Yaskawa INFORM job: A_ROOF_UPPER_0614_2_PAINT_35.JBI

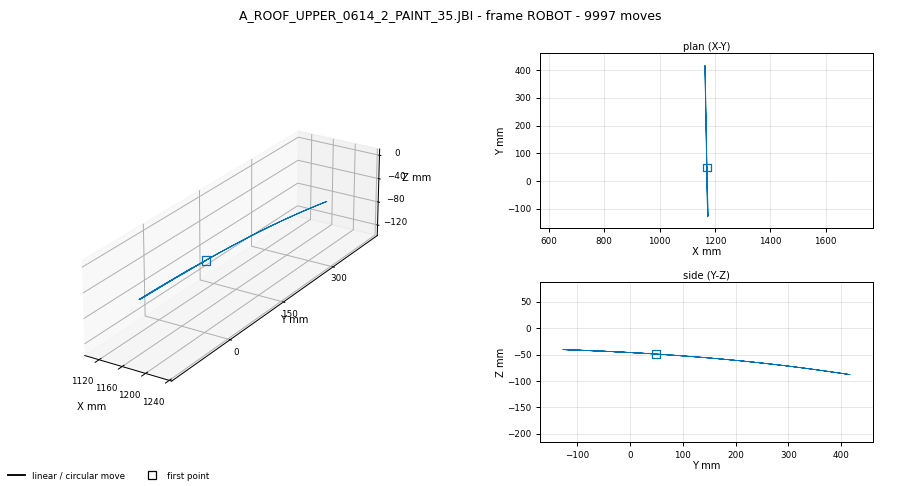
[picture p0: tool path of A_ROOF_UPPER_0614_2_PAINT_35.JBI in frame ROBOT, 9997 of 9997 moves have a stored position in this frame; points joined in program order, loops and branches not executed]
/JOB
//NAME A_ROOF_UPPER_0614_2_PAINT35
//POS
///NPOS 9997,0,0,0,0,0
///TOOL 1
///USER 0
///POSTYPE ROBOT
///RECTAN
///RCONF 1,0,0,0,0,0,0,0,0,0,0,0,0,0,0,0,0,0,0,0,0,0,0,0
C00000=1171.843,48.979,-48.682,-179.550,6.056,148.954
C00001=1171.848,48.730,-48.666,-179.552,6.054,148.954
C00002=1171.853,48.480,-48.650,-179.555,6.054,148.955
C00003=1171.858,48.231,-48.635,-179.557,6.053,148.955
C00004=1171.863,47.981,-48.619,-179.560,6.052,148.956
C00005=1171.868,47.732,-48.604,-179.562,6.051,148.956
C00006=1171.873,47.482,-48.588,-179.565,6.050,148.957
C00007=1171.878,47.233,-48.571,-179.568,6.049,148.958
C00008=1171.882,46.984,-48.556,-179.570,6.048,148.958
C00009=1171.888,46.734,-48.541,-179.573,6.048,148.959
C00010=1171.893,46.484,-48.525,-179.575,6.047,148.959
C00011=1171.898,46.235,-48.509,-179.578,6.046,148.960
C00012=1171.903,45.986,-48.494,-179.581,6.045,148.960
C00013=1171.908,45.736,-48.479,-179.583,6.044,148.961
C00014=1171.913,45.487,-48.462,-179.586,6.043,148.962
C00015=1171.918,45.237,-48.446,-179.589,6.042,148.962
C00016=1171.923,44.988,-48.431,-179.591,6.041,148.963
C00017=1171.927,44.738,-48.415,-179.593,6.041,148.963
C00018=1171.933,44.489,-48.400,-179.597,6.039,148.964
C00019=1171.938,44.239,-48.384,-179.599,6.038,148.964
C00020=1171.943,43.990,-48.369,-179.601,6.038,148.965
C00021=1171.948,43.740,-48.353,-179.604,6.036,148.966
C00022=1171.953,43.491,-48.338,-179.607,6.036,148.966
C00023=1171.958,43.242,-48.323,-179.609,6.035,148.967
C00024=1171.963,42.992,-48.307,-179.612,6.034,148.967
C00025=1171.968,42.742,-48.291,-179.614,6.033,148.968
C00026=1171.972,42.493,-48.276,-179.617,6.032,148.968
C00027=1171.978,42.244,-48.261,-179.620,6.032,148.969
C00028=1171.983,41.994,-48.245,-179.622,6.031,148.970
C00029=1171.988,41.745,-48.230,-179.625,6.030,148.970
C00030=1171.993,41.495,-48.214,-179.627,6.029,148.971
C00031=1171.998,41.246,-48.199,-179.630,6.028,148.971
C00032=1172.003,40.997,-48.184,-179.633,6.027,148.972
C00033=1172.008,40.747,-48.168,-179.635,6.026,148.972
C00034=1172.012,40.497,-48.153,-179.637,6.025,148.973
C00035=1172.018,40.247,-48.138,-179.640,6.025,148.974
C00036=1172.023,39.998,-48.122,-179.643,6.023,148.974
C00037=1172.028,39.749,-48.107,-179.645,6.023,148.975
C00038=1172.033,39.499,-48.092,-179.648,6.022,148.975
C00039=1172.039,39.250,-48.076,-179.650,6.021,148.976
C00040=1172.043,39.000,-48.061,-179.653,6.020,148.977
C00041=1172.048,38.751,-48.045,-179.656,6.019,148.977
C00042=1172.053,38.502,-48.030,-179.658,6.019,148.978
C00043=1172.058,38.252,-48.015,-179.661,6.018,148.978
C00044=1172.063,38.003,-48.000,-179.664,6.016,148.979
C00045=1172.068,37.753,-47.985,-179.666,6.016,148.979
C00046=1172.072,37.503,-47.969,-179.668,6.015,148.980
C00047=1172.078,37.254,-47.954,-179.671,6.015,148.981
C00048=1172.084,37.004,-47.939,-179.674,6.013,148.981
C00049=1172.088,36.755,-47.924,-179.677,6.012,148.982
C00050=1172.094,36.505,-47.908,-179.679,6.012,148.982
C00051=1172.098,36.256,-47.893,-179.681,6.011,148.983
C00052=1172.104,36.007,-47.878,-179.684,6.011,148.983
C00053=1172.109,35.757,-47.863,-179.687,6.009,148.984
C00054=1172.113,35.507,-47.847,-179.689,6.008,148.985
C00055=1172.118,35.258,-47.832,-179.691,6.008,148.985
C00056=1172.124,35.008,-47.817,-179.694,6.007,148.986
C00057=1172.128,34.759,-47.802,-179.697,6.006,148.986
C00058=1172.134,34.510,-47.787,-179.700,6.005,148.987
C00059=1172.138,34.260,-47.772,-179.702,6.004,148.988
C00060=1172.144,34.010,-47.757,-179.704,6.004,148.988
C00061=1172.149,33.761,-47.742,-179.707,6.003,148.989
C00062=1172.153,33.512,-47.727,-179.710,6.002,148.989
C00063=1172.159,33.262,-47.712,-179.712,6.001,148.990
C00064=1172.163,33.012,-47.697,-179.715,6.000,148.990
C00065=1172.169,32.763,-47.681,-179.717,6.000,148.991
C00066=1172.173,32.513,-47.667,-179.720,5.998,148.992
C00067=1172.179,32.264,-47.651,-179.723,5.997,148.992
C00068=1172.184,32.014,-47.637,-179.725,5.997,148.993
C00069=1172.188,31.765,-47.622,-179.728,5.996,148.993
C00070=1172.194,31.516,-47.607,-179.730,5.996,148.994
C00071=1172.199,31.266,-47.592,-179.733,5.994,148.994
C00072=1172.203,31.017,-47.577,-179.735,5.993,148.995
C00073=1172.209,30.767,-47.562,-179.738,5.993,148.996
C00074=1172.214,30.518,-47.547,-179.741,5.992,148.996
C00075=1172.219,30.268,-47.533,-179.743,5.992,148.997
C00076=1172.224,30.019,-47.518,-179.746,5.990,148.997
C00077=1172.229,29.769,-47.503,-179.748,5.989,148.998
C00078=1172.234,29.520,-47.488,-179.751,5.989,148.999
C00079=1172.239,29.271,-47.473,-179.754,5.988,148.999
C00080=1172.244,29.021,-47.458,-179.756,5.988,149.000
C00081=1172.249,28.771,-47.443,-179.759,5.986,149.000
C00082=1172.255,28.503,-47.427,-179.762,5.986,149.001
C00083=1172.260,28.234,-47.411,-179.764,5.985,149.001
C00084=1172.266,27.965,-47.395,-179.767,5.984,149.002
C00085=1172.271,27.696,-47.379,-179.770,5.983,149.003
C00086=1172.276,27.446,-47.365,-179.772,5.983,149.004
C00087=1172.281,27.197,-47.350,-179.774,5.982,149.004
C00088=1172.286,26.947,-47.335,-179.777,5.981,149.005
C00089=1172.291,26.697,-47.321,-179.780,5.980,149.005
C00090=1172.296,26.448,-47.305,-179.782,5.979,149.006
C00091=1172.301,26.198,-47.291,-179.785,5.979,149.006
C00092=1172.306,25.949,-47.276,-179.787,5.978,149.007
C00093=1172.311,25.699,-47.262,-179.790,5.977,149.008
C00094=1172.317,25.449,-47.247,-179.792,5.977,149.008
C00095=1172.321,25.200,-47.232,-179.795,5.975,149.009
C00096=1172.326,24.951,-47.218,-179.798,5.975,149.009
C00097=1172.331,24.702,-47.203,-179.800,5.974,149.010
C00098=1172.337,24.452,-47.188,-179.803,5.974,149.011
C00099=1172.342,24.203,-47.174,-179.805,5.973,149.011
C00100=1172.347,23.953,-47.159,-179.808,5.972,149.012
C00101=1172.352,23.704,-47.145,-179.811,5.971,149.012
C00102=1172.357,23.454,-47.130,-179.813,5.970,149.013
C00103=1172.362,23.204,-47.115,-179.816,5.970,149.013
C00104=1172.367,22.955,-47.100,-179.818,5.969,149.014
C00105=1172.372,22.705,-47.086,-179.820,5.968,149.015
C00106=1172.377,22.455,-47.072,-179.823,5.968,149.015
C00107=1172.382,22.206,-47.057,-179.826,5.966,149.016
C00108=1172.386,21.957,-47.043,-179.829,5.966,149.016
C00109=1172.392,21.707,-47.028,-179.831,5.965,149.017
C00110=1172.398,21.458,-47.014,-179.833,5.964,149.018
C00111=1172.402,21.209,-46.999,-179.836,5.964,149.018
C00112=1172.407,20.959,-46.985,-179.838,5.963,149.019
C00113=1172.412,20.709,-46.970,-179.841,5.962,149.019
C00114=1172.417,20.459,-46.956,-179.844,5.961,149.020
C00115=1172.422,20.210,-46.942,-179.846,5.960,149.021
C00116=1172.427,19.961,-46.927,-179.849,5.960,149.021
C00117=1172.433,19.711,-46.912,-179.851,5.959,149.022
C00118=1172.438,19.462,-46.898,-179.854,5.959,149.022
C00119=1172.443,19.212,-46.884,-179.856,5.958,149.023
C00120=1172.448,18.962,-46.869,-179.858,5.957,149.023
C00121=1172.453,18.712,-46.855,-179.862,5.956,149.024
C00122=1172.458,18.463,-46.840,-179.864,5.955,149.025
C00123=1172.463,18.214,-46.826,-179.867,5.955,149.025
C00124=1172.468,17.965,-46.812,-179.869,5.954,149.026
C00125=1172.473,17.715,-46.798,-179.871,5.953,149.026
C00126=1172.478,17.465,-46.783,-179.874,5.953,149.027
C00127=1172.483,17.216,-46.769,-179.876,5.952,149.028
C00128=1172.488,16.966,-46.755,-179.879,5.951,149.028
C00129=1172.493,16.716,-46.741,-179.881,5.951,149.029
C00130=1172.498,16.467,-46.727,-179.884,5.949,149.029
C00131=1172.503,16.217,-46.712,-179.887,5.949,149.030
C00132=1172.508,15.968,-46.698,-179.889,5.948,149.031
C00133=1172.513,15.719,-46.683,-179.892,5.948,149.031
C00134=1172.518,15.469,-46.669,-179.894,5.947,149.032
C00135=1172.524,15.220,-46.655,-179.896,5.946,149.032
C00136=1172.528,14.970,-46.641,-179.899,5.946,149.033
C00137=1172.533,14.720,-46.626,-179.902,5.945,149.034
C00138=1172.538,14.471,-46.612,-179.904,5.944,149.034
C00139=1172.544,14.222,-46.598,-179.907,5.943,149.035
C00140=1172.549,13.972,-46.584,-179.909,5.942,149.035
C00141=1172.554,13.722,-46.570,-179.912,5.942,149.036
C00142=1172.559,13.473,-46.555,-179.915,5.941,149.037
C00143=1172.565,13.223,-46.542,-179.917,5.941,149.037
C00144=1172.570,12.973,-46.528,-179.919,5.940,149.038
C00145=1172.575,12.724,-46.514,-179.922,5.940,149.038
C00146=1172.580,12.474,-46.499,-179.924,5.939,149.039
C00147=1172.585,12.225,-46.485,-179.927,5.938,149.040
C00148=1172.590,11.975,-46.471,-179.929,5.937,149.040
C00149=1172.595,11.725,-46.457,-179.932,5.936,149.041
C00150=1172.600,11.476,-46.443,-179.935,5.936,149.041
C00151=1172.606,11.227,-46.429,-179.937,5.935,149.042
C00152=1172.610,10.977,-46.415,-179.940,5.934,149.043
C00153=1172.615,10.728,-46.401,-179.942,5.934,149.043
C00154=1172.620,10.477,-46.387,-179.945,5.933,149.044
C00155=1172.626,10.228,-46.373,-179.947,5.933,149.044
C00156=1172.630,9.979,-46.359,-179.949,5.932,149.045
C00157=1172.635,9.729,-46.345,-179.952,5.931,149.046
C00158=1172.641,9.480,-46.331,-179.955,5.931,149.046
C00159=1172.646,9.230,-46.317,-179.957,5.930,149.047
C00160=1172.650,8.980,-46.304,-179.960,5.929,149.047
C00161=1172.656,8.731,-46.290,-179.963,5.928,149.048
C00162=1172.661,8.481,-46.275,-179.965,5.927,149.049
C00163=1172.666,8.232,-46.261,-179.968,5.927,149.049
C00164=1172.671,7.983,-46.247,-179.970,5.926,149.050
C00165=1172.676,7.733,-46.234,-179.972,5.926,149.050
C00166=1172.681,7.483,-46.220,-179.975,5.925,149.051
C00167=1172.687,7.234,-46.206,-179.977,5.924,149.052
C00168=1172.691,6.984,-46.192,-179.980,5.924,149.052
C00169=1172.697,6.734,-46.178,-179.983,5.923,149.053
C00170=1172.702,6.485,-46.165,-179.985,5.923,149.053
C00171=1172.706,6.235,-46.151,-179.987,5.922,149.054
C00172=1172.711,5.986,-46.136,-179.990,5.921,149.054
C00173=1172.717,5.736,-46.123,-179.992,5.921,149.055
C00174=1172.722,5.486,-46.109,-179.995,5.920,149.056
C00175=1172.726,5.237,-46.095,-179.997,5.919,149.056
C00176=1172.732,4.987,-46.082,-180.000,5.919,149.057
C00177=1172.737,4.738,-46.068,179.997,5.918,149.058
C00178=1172.743,4.489,-46.054,179.995,5.917,149.058
C00179=1172.747,4.239,-46.041,179.992,5.916,149.059
C00180=1172.752,3.989,-46.027,179.990,5.916,149.059
C00181=1172.758,3.740,-46.013,179.987,5.915,149.060
C00182=1172.762,3.490,-46.000,179.985,5.915,149.061
C00183=1172.768,3.241,-45.986,179.983,5.914,149.061
C00184=1172.773,2.991,-45.972,179.980,5.913,149.062
C00185=1172.778,2.741,-45.958,179.977,5.913,149.063
C00186=1172.783,2.472,-45.944,179.975,5.912,149.063
C00187=1172.789,2.203,-45.929,179.972,5.912,149.064
C00188=1172.794,1.934,-45.914,179.970,5.911,149.064
C00189=1172.800,1.664,-45.899,179.967,5.910,149.065
C00190=1172.806,1.415,-45.886,179.964,5.909,149.066
C00191=1172.810,1.165,-45.872,179.962,5.909,149.066
C00192=1172.816,0.916,-45.859,179.959,5.908,149.067
C00193=1172.821,0.666,-45.845,179.956,5.908,149.068
C00194=1172.826,0.417,-45.832,179.954,5.907,149.068
C00195=1172.831,0.167,-45.818,179.952,5.906,149.069
C00196=1172.835,-0.083,-45.805,179.949,5.905,149.069
C00197=1172.841,-0.332,-45.791,179.947,5.905,149.070
C00198=1172.846,-0.583,-45.777,179.944,5.905,149.071
C00199=1172.851,-0.831,-45.764,179.942,5.904,149.071
C00200=1172.856,-1.082,-45.750,179.939,5.903,149.072
C00201=1172.862,-1.331,-45.736,179.937,5.903,149.072
C00202=1172.866,-1.581,-45.723,179.934,5.902,149.073
C00203=1172.872,-1.830,-45.710,179.932,5.902,149.074
C00204=1172.876,-2.080,-45.697,179.929,5.901,149.074
C00205=1172.882,-2.329,-45.683,179.927,5.900,149.075
C00206=1172.886,-2.579,-45.670,179.924,5.900,149.075
C00207=1172.892,-2.828,-45.657,179.922,5.899,149.076
C00208=1172.897,-3.078,-45.642,179.920,5.898,149.077
C00209=1172.902,-3.327,-45.630,179.917,5.898,149.077
C00210=1172.907,-3.577,-45.615,179.915,5.897,149.078
C00211=1172.912,-3.826,-45.603,179.912,5.897,149.078
C00212=1172.918,-4.077,-45.589,179.909,5.896,149.079
C00213=1172.923,-4.325,-45.576,179.907,5.895,149.080
C00214=1172.928,-4.576,-45.562,179.905,5.895,149.080
C00215=1172.933,-4.825,-45.550,179.902,5.895,149.081
C00216=1172.938,-5.075,-45.535,179.900,5.894,149.081
C00217=1172.943,-5.324,-45.523,179.897,5.893,149.082
C00218=1172.948,-5.574,-45.509,179.895,5.892,149.083
C00219=1172.953,-5.823,-45.496,179.892,5.892,149.083
C00220=1172.959,-6.073,-45.483,179.890,5.891,149.084
C00221=1172.963,-6.323,-45.470,179.887,5.891,149.084
C00222=1172.969,-6.572,-45.456,179.885,5.890,149.085
C00223=1172.974,-6.822,-45.443,179.882,5.890,149.086
C00224=1172.979,-7.071,-45.430,179.880,5.889,149.086
C00225=1172.984,-7.321,-45.417,179.877,5.888,149.087
C00226=1172.989,-7.570,-45.403,179.875,5.888,149.088
C00227=1172.994,-7.820,-45.390,179.872,5.887,149.088
C00228=1173.000,-8.070,-45.377,179.870,5.887,149.089
C00229=1173.005,-8.319,-45.364,179.867,5.886,149.089
C00230=1173.009,-8.569,-45.350,179.865,5.885,149.090
C00231=1173.015,-8.818,-45.337,179.862,5.885,149.091
C00232=1173.020,-9.068,-45.324,179.860,5.884,149.091
C00233=1173.025,-9.318,-45.311,179.857,5.884,149.092
C00234=1173.030,-9.567,-45.298,179.855,5.883,149.092
C00235=1173.035,-9.817,-45.285,179.853,5.882,149.093
C00236=1173.041,-10.066,-45.272,179.850,5.882,149.094
C00237=1173.045,-10.316,-45.259,179.847,5.881,149.094
C00238=1173.051,-10.566,-45.245,179.845,5.881,149.095
C00239=1173.056,-10.815,-45.233,179.842,5.880,149.095
C00240=1173.060,-11.065,-45.219,179.840,5.880,149.096
C00241=1173.066,-11.314,-45.206,179.838,5.879,149.097
C00242=1173.071,-11.564,-45.193,179.835,5.878,149.097
C00243=1173.076,-11.814,-45.180,179.833,5.879,149.098
C00244=1173.082,-12.063,-45.167,179.831,5.878,149.098
C00245=1173.086,-12.313,-45.154,179.828,5.878,149.099
C00246=1173.091,-12.563,-45.142,179.826,5.877,149.100
C00247=1173.097,-12.812,-45.128,179.823,5.876,149.100
C00248=1173.102,-13.062,-45.115,179.821,5.876,149.101
C00249=1173.107,-13.311,-45.102,179.818,5.875,149.101
C00250=1173.112,-13.561,-45.089,179.816,5.875,149.102
C00251=1173.117,-13.811,-45.076,179.813,5.874,149.103
C00252=1173.122,-14.060,-45.063,179.811,5.873,149.103
C00253=1173.128,-14.310,-45.050,179.808,5.873,149.104
C00254=1173.132,-14.560,-45.037,179.806,5.872,149.105
C00255=1173.138,-14.809,-45.025,179.803,5.872,149.105
C00256=1173.143,-15.059,-45.011,179.801,5.871,149.106
C00257=1173.148,-15.309,-44.998,179.798,5.871,149.107
C00258=1173.153,-15.558,-44.986,179.796,5.870,149.107
C00259=1173.158,-15.807,-44.973,179.793,5.869,149.108
C00260=1173.164,-16.057,-44.960,179.791,5.869,149.108
C00261=1173.169,-16.307,-44.947,179.788,5.868,149.109
C00262=1173.174,-16.556,-44.934,179.786,5.868,149.110
C00263=1173.179,-16.806,-44.922,179.784,5.868,149.110
C00264=1173.184,-17.056,-44.908,179.782,5.867,149.111
C00265=1173.189,-17.305,-44.896,179.779,5.867,149.111
C00266=1173.194,-17.554,-44.883,179.777,5.866,149.112
C00267=1173.199,-17.804,-44.871,179.774,5.865,149.113
C00268=1173.205,-18.055,-44.858,179.771,5.865,149.113
C00269=1173.210,-18.304,-44.845,179.769,5.864,149.114
C00270=1173.215,-18.553,-44.832,179.767,5.864,149.114
C00271=1173.220,-18.803,-44.819,179.764,5.863,149.115
C00272=1173.225,-19.053,-44.807,179.762,5.862,149.116
C00273=1173.231,-19.302,-44.794,179.759,5.862,149.116
C00274=1173.236,-19.552,-44.781,179.757,5.861,149.117
C00275=1173.241,-19.801,-44.768,179.754,5.861,149.117
C00276=1173.246,-20.051,-44.756,179.752,5.860,149.118
C00277=1173.251,-20.301,-44.744,179.750,5.860,149.119
C00278=1173.256,-20.550,-44.731,179.747,5.860,149.119
C00279=1173.262,-20.800,-44.718,179.745,5.859,149.120
C00280=1173.267,-21.050,-44.705,179.742,5.859,149.121
C00281=1173.272,-21.299,-44.692,179.740,5.858,149.121
C00282=1173.277,-21.549,-44.680,179.737,5.858,149.122
C00283=1173.282,-21.798,-44.668,179.735,5.857,149.122
C00284=1173.287,-22.048,-44.655,179.732,5.856,149.123
C00285=1173.292,-22.298,-44.642,179.730,5.856,149.124
C00286=1173.298,-22.547,-44.629,179.727,5.855,149.124
C00287=1173.303,-22.797,-44.617,179.725,5.855,149.125
C00288=1173.308,-23.047,-44.605,179.723,5.855,149.125
C00289=1173.313,-23.296,-44.592,179.721,5.854,149.126
C00290=1173.318,-23.566,-44.578,179.718,5.854,149.127
C00291=1173.324,-23.836,-44.565,179.715,5.853,149.127
C00292=1173.330,-24.105,-44.551,179.713,5.853,149.128
C00293=1173.335,-24.375,-44.538,179.710,5.851,149.129
C00294=1173.340,-24.625,-44.526,179.708,5.852,149.129
C00295=1173.346,-24.874,-44.513,179.705,5.851,149.130
C00296=1173.350,-25.124,-44.500,179.703,5.850,149.131
C00297=1173.356,-25.374,-44.487,179.700,5.850,149.131
C00298=1173.361,-25.624,-44.475,179.698,5.849,149.132
C00299=1173.367,-25.873,-44.463,179.695,5.849,149.132
C00300=1173.372,-26.123,-44.450,179.693,5.848,149.133
C00301=1173.377,-26.373,-44.438,179.690,5.848,149.134
C00302=1173.382,-26.622,-44.425,179.688,5.847,149.134
C00303=1173.387,-26.872,-44.413,179.686,5.847,149.135
C00304=1173.392,-27.122,-44.401,179.683,5.847,149.136
C00305=1173.397,-27.371,-44.388,179.681,5.846,149.136
C00306=1173.403,-27.621,-44.376,179.678,5.846,149.137
C00307=1173.408,-27.870,-44.364,179.676,5.845,149.137
C00308=1173.413,-28.120,-44.351,179.674,5.844,149.138
C00309=1173.418,-28.370,-44.339,179.671,5.844,149.139
C00310=1173.424,-28.619,-44.326,179.669,5.843,149.139
C00311=1173.428,-28.870,-44.314,179.667,5.843,149.140
C00312=1173.433,-29.119,-44.302,179.664,5.843,149.141
C00313=1173.439,-29.368,-44.289,179.662,5.842,149.141
C00314=1173.443,-29.618,-44.278,179.659,5.842,149.142
C00315=1173.448,-29.867,-44.265,179.656,5.841,149.142
C00316=1173.454,-30.117,-44.253,179.654,5.841,149.143
C00317=1173.459,-30.366,-44.241,179.652,5.840,149.144
C00318=1173.464,-30.616,-44.229,179.649,5.840,149.144
C00319=1173.469,-30.866,-44.216,179.647,5.840,149.145
C00320=1173.475,-31.116,-44.204,179.645,5.839,149.145
C00321=1173.480,-31.365,-44.192,179.643,5.838,149.146
C00322=1173.485,-31.616,-44.179,179.640,5.838,149.147
C00323=1173.490,-31.865,-44.167,179.637,5.837,149.147
C00324=1173.495,-32.115,-44.155,179.635,5.837,149.148
C00325=1173.501,-32.364,-44.142,179.632,5.836,149.148
C00326=1173.506,-32.614,-44.130,179.630,5.837,149.149
C00327=1173.510,-32.863,-44.118,179.628,5.836,149.150
C00328=1173.516,-33.113,-44.107,179.625,5.835,149.150
C00329=1173.521,-33.362,-44.094,179.623,5.835,149.151
C00330=1173.526,-33.612,-44.082,179.621,5.834,149.152
C00331=1173.532,-33.862,-44.070,179.618,5.834,149.152
C00332=1173.537,-34.112,-44.058,179.616,5.833,149.153
C00333=1173.542,-34.362,-44.046,179.614,5.833,149.153
C00334=1173.547,-34.611,-44.034,179.611,5.833,149.154
C00335=1173.552,-34.860,-44.022,179.609,5.832,149.155
C00336=1173.558,-35.110,-44.010,179.606,5.832,149.155
C00337=1173.563,-35.360,-43.997,179.603,5.831,149.156
C00338=1173.568,-35.610,-43.985,179.601,5.830,149.156
C00339=1173.573,-35.859,-43.973,179.599,5.831,149.157
C00340=1173.578,-36.109,-43.962,179.597,5.830,149.158
C00341=1173.583,-36.359,-43.950,179.594,5.829,149.158
C00342=1173.589,-36.608,-43.937,179.592,5.829,149.159
C00343=1173.594,-36.858,-43.925,179.590,5.828,149.159
C00344=1173.599,-37.108,-43.913,179.587,5.828,149.160
C00345=1173.604,-37.357,-43.901,179.585,5.828,149.161
C00346=1173.609,-37.607,-43.889,179.583,5.827,149.161
C00347=1173.615,-37.857,-43.878,179.580,5.827,149.162
C00348=1173.620,-38.106,-43.865,179.577,5.826,149.163
C00349=1173.625,-38.356,-43.853,179.575,5.826,149.163
C00350=1173.630,-38.605,-43.842,179.572,5.825,149.164
C00351=1173.635,-38.855,-43.830,179.571,5.825,149.164
C00352=1173.640,-39.105,-43.817,179.568,5.825,149.165
C00353=1173.646,-39.355,-43.805,179.566,5.824,149.166
C00354=1173.651,-39.604,-43.794,179.563,5.823,149.166
C00355=1173.657,-39.854,-43.783,179.561,5.823,149.167
C00356=1173.662,-40.103,-43.770,179.558,5.823,149.168
C00357=1173.667,-40.353,-43.758,179.556,5.823,149.168
C00358=1173.672,-40.602,-43.747,179.554,5.822,149.169
C00359=1173.677,-40.852,-43.735,179.551,5.822,149.170
C00360=1173.683,-41.102,-43.723,179.549,5.821,149.170
C00361=1173.687,-41.351,-43.711,179.546,5.821,149.171
C00362=1173.692,-41.601,-43.699,179.545,5.820,149.171
C00363=1173.698,-41.851,-43.687,179.542,5.820,149.172
C00364=1173.703,-42.101,-43.676,179.539,5.820,149.173
C00365=1173.708,-42.351,-43.664,179.537,5.819,149.173
C00366=1173.713,-42.600,-43.651,179.534,5.818,149.174
C00367=1173.718,-42.850,-43.640,179.532,5.818,149.174
C00368=1173.724,-43.099,-43.629,179.530,5.818,149.175
C00369=1173.729,-43.349,-43.617,179.528,5.818,149.176
C00370=1173.734,-43.598,-43.605,179.525,5.817,149.176
C00371=1173.739,-43.848,-43.594,179.523,5.816,149.177
C00372=1173.745,-44.098,-43.582,179.520,5.816,149.178
C00373=1173.750,-44.348,-43.570,179.518,5.816,149.178
C00374=1173.755,-44.597,-43.558,179.516,5.815,149.179
C00375=1173.760,-44.847,-43.546,179.513,5.815,149.179
C00376=1173.765,-45.096,-43.535,179.511,5.814,149.180
C00377=1173.771,-45.346,-43.523,179.508,5.814,149.181
C00378=1173.776,-45.596,-43.512,179.507,5.814,149.181
C00379=1173.781,-45.846,-43.500,179.504,5.813,149.182
C00380=1173.786,-46.096,-43.488,179.501,5.813,149.182
C00381=1173.791,-46.345,-43.477,179.499,5.812,149.183
C00382=1173.796,-46.595,-43.465,179.497,5.812,149.184
C00383=1173.802,-46.844,-43.454,179.494,5.812,149.184
C00384=1173.807,-47.094,-43.442,179.492,5.811,149.185
C00385=1173.812,-47.344,-43.431,179.490,5.811,149.186
C00386=1173.817,-47.594,-43.419,179.487,5.810,149.186
C00387=1173.823,-47.844,-43.407,179.485,5.810,149.187
C00388=1173.827,-48.093,-43.396,179.483,5.810,149.187
C00389=1173.833,-48.342,-43.384,179.480,5.809,149.188
C00390=1173.838,-48.592,-43.373,179.478,5.809,149.189
C00391=1173.844,-48.842,-43.361,179.476,5.808,149.189
C00392=1173.848,-49.092,-43.350,179.474,5.808,149.190
C00393=1173.854,-49.341,-43.338,179.471,5.808,149.190
C00394=1173.860,-49.612,-43.326,179.468,5.807,149.191
C00395=1173.865,-49.882,-43.313,179.466,5.807,149.192
C00396=1173.871,-50.153,-43.301,179.463,5.806,149.192
C00397=1173.877,-50.423,-43.288,179.461,5.806,149.193
C00398=1173.881,-50.672,-43.277,179.458,5.805,149.194
C00399=1173.887,-50.922,-43.265,179.456,5.805,149.194
C00400=1173.892,-51.172,-43.254,179.454,5.805,149.195
C00401=1173.898,-51.421,-43.242,179.451,5.805,149.196
C00402=1173.903,-51.671,-43.232,179.449,5.804,149.196
C00403=1173.908,-51.921,-43.220,179.447,5.804,149.197
C00404=1173.913,-52.171,-43.208,179.445,5.803,149.197
C00405=1173.918,-52.420,-43.197,179.442,5.803,149.198
C00406=1173.923,-52.670,-43.186,179.439,5.802,149.199
C00407=1173.928,-52.919,-43.174,179.438,5.802,149.199
C00408=1173.934,-53.169,-43.162,179.435,5.802,149.200
C00409=1173.939,-53.419,-43.152,179.433,5.801,149.200
C00410=1173.945,-53.669,-43.140,179.430,5.801,149.201
C00411=1173.949,-53.919,-43.129,179.428,5.801,149.202
C00412=1173.955,-54.168,-43.117,179.426,5.800,149.202
C00413=1173.960,-54.417,-43.106,179.423,5.800,149.203
C00414=1173.965,-54.667,-43.095,179.421,5.799,149.203
C00415=1173.970,-54.918,-43.084,179.419,5.800,149.204
C00416=1173.975,-55.167,-43.072,179.416,5.799,149.205
C00417=1173.980,-55.416,-43.062,179.414,5.798,149.205
C00418=1173.986,-55.666,-43.050,179.412,5.798,149.206
C00419=1173.991,-55.916,-43.039,179.409,5.798,149.207
C00420=1173.997,-56.166,-43.028,179.407,5.797,149.207
C00421=1174.002,-56.415,-43.016,179.405,5.797,149.208
C00422=1174.006,-56.665,-43.005,179.402,5.796,149.208
C00423=1174.012,-56.915,-42.994,179.400,5.797,149.209
C00424=1174.017,-57.164,-42.983,179.398,5.796,149.210
C00425=1174.022,-57.414,-42.972,179.395,5.795,149.210
C00426=1174.027,-57.664,-42.960,179.393,5.795,149.211
C00427=1174.033,-57.913,-42.950,179.391,5.795,149.211
C00428=1174.038,-58.163,-42.938,179.389,5.795,149.212
C00429=1174.043,-58.413,-42.926,179.386,5.794,149.213
C00430=1174.049,-58.662,-42.916,179.384,5.793,149.213
C00431=1174.053,-58.912,-42.905,179.382,5.794,149.214
C00432=1174.059,-59.162,-42.893,179.379,5.793,149.214
C00433=1174.064,-59.412,-42.883,179.377,5.793,149.215
C00434=1174.069,-59.661,-42.871,179.374,5.792,149.216
C00435=1174.075,-59.911,-42.860,179.373,5.792,149.216
C00436=1174.080,-60.161,-42.849,179.370,5.792,149.217
C00437=1174.085,-60.410,-42.838,179.368,5.791,149.218
C00438=1174.090,-60.660,-42.827,179.366,5.791,149.218
C00439=1174.096,-60.910,-42.816,179.363,5.791,149.219
C00440=1174.101,-61.159,-42.805,179.361,5.790,149.219
C00441=1174.106,-61.410,-42.794,179.358,5.790,149.220
C00442=1174.112,-61.659,-42.783,179.356,5.790,149.221
C00443=1174.116,-61.909,-42.771,179.354,5.789,149.221
C00444=1174.121,-62.159,-42.761,179.351,5.789,149.222
C00445=1174.127,-62.408,-42.750,179.349,5.788,149.223
C00446=1174.132,-62.658,-42.739,179.347,5.788,149.223
C00447=1174.138,-62.907,-42.728,179.345,5.788,149.224
C00448=1174.143,-63.157,-42.717,179.342,5.787,149.224
C00449=1174.147,-63.407,-42.706,179.340,5.788,149.225
C00450=1174.153,-63.657,-42.696,179.338,5.787,149.226
C00451=1174.158,-63.907,-42.684,179.335,5.786,149.226
C00452=1174.164,-64.155,-42.673,179.333,5.786,149.227
C00453=1174.169,-64.406,-42.662,179.331,5.786,149.227
C00454=1174.173,-64.655,-42.651,179.329,5.785,149.228
C00455=1174.179,-64.905,-42.641,179.326,5.785,149.229
C00456=1174.184,-65.155,-42.629,179.324,5.785,149.229
C00457=1174.190,-65.404,-42.619,179.322,5.784,149.230
C00458=1174.195,-65.654,-42.607,179.319,5.784,149.231
C00459=1174.200,-65.904,-42.597,179.317,5.784,149.231
C00460=1174.205,-66.154,-42.587,179.315,5.784,149.232
C00461=1174.211,-66.404,-42.575,179.312,5.783,149.232
C00462=1174.216,-66.653,-42.565,179.310,5.782,149.233
C00463=1174.221,-66.903,-42.553,179.308,5.783,149.234
C00464=1174.227,-67.152,-42.543,179.306,5.782,149.234
C00465=1174.231,-67.402,-42.532,179.303,5.782,149.235
C00466=1174.237,-67.652,-42.522,179.301,5.782,149.235
C00467=1174.242,-67.902,-42.511,179.299,5.781,149.236
C00468=1174.247,-68.152,-42.499,179.296,5.781,149.237
C00469=1174.253,-68.401,-42.489,179.294,5.781,149.237
C00470=1174.258,-68.651,-42.478,179.292,5.780,149.238
C00471=1174.263,-68.900,-42.467,179.290,5.779,149.238
C00472=1174.268,-69.151,-42.457,179.287,5.779,149.239
C00473=1174.273,-69.400,-42.446,179.285,5.779,149.240
C00474=1174.278,-69.650,-42.435,179.283,5.779,149.240
C00475=1174.284,-69.899,-42.424,179.280,5.778,149.241
C00476=1174.289,-70.149,-42.413,179.278,5.778,149.241
C00477=1174.295,-70.399,-42.403,179.276,5.778,149.242
C00478=1174.300,-70.649,-42.392,179.274,5.777,149.243
C00479=1174.305,-70.898,-42.381,179.271,5.777,149.243
C00480=1174.310,-71.148,-42.371,179.269,5.777,149.244
C00481=1174.316,-71.397,-42.360,179.267,5.776,149.245
C00482=1174.321,-71.647,-42.349,179.265,5.777,149.245
C00483=1174.326,-71.897,-42.339,179.262,5.776,149.246
C00484=1174.331,-72.147,-42.329,179.260,5.775,149.246
C00485=1174.337,-72.396,-42.318,179.258,5.775,149.247
C00486=1174.342,-72.646,-42.307,179.255,5.775,149.248
C00487=1174.347,-72.896,-42.297,179.253,5.775,149.248
C00488=1174.352,-73.146,-42.286,179.251,5.775,149.249
C00489=1174.357,-73.395,-42.275,179.248,5.774,149.250
C00490=1174.363,-73.645,-42.265,179.246,5.773,149.250
C00491=1174.368,-73.895,-42.255,179.244,5.774,149.251
C00492=1174.374,-74.144,-42.244,179.242,5.773,149.251
C00493=1174.378,-74.394,-42.233,179.239,5.773,149.252
C00494=1174.384,-74.644,-42.223,179.237,5.773,149.253
C00495=1174.389,-74.894,-42.212,179.235,5.772,149.253
C00496=1174.395,-75.143,-42.202,179.232,5.772,149.254
C00497=1174.399,-75.393,-42.191,179.231,5.772,149.254
C00498=1174.406,-75.664,-42.180,179.228,5.771,149.255
C00499=1174.412,-75.936,-42.168,179.225,5.771,149.256
C00500=1174.417,-76.207,-42.157,179.223,5.771,149.256
C00501=1174.423,-76.477,-42.145,179.221,5.770,149.257
C00502=1174.428,-76.727,-42.135,179.219,5.770,149.258
C00503=1174.434,-76.977,-42.125,179.216,5.769,149.258
C00504=1174.439,-77.226,-42.114,179.214,5.769,149.259
C00505=1174.444,-77.477,-42.104,179.212,5.769,149.260
C00506=1174.450,-77.726,-42.094,179.209,5.769,149.260
C00507=1174.454,-77.976,-42.083,179.207,5.768,149.261
C00508=1174.459,-78.225,-42.073,179.205,5.768,149.261
C00509=1174.465,-78.475,-42.062,179.202,5.768,149.262
C00510=1174.470,-78.725,-42.052,179.200,5.767,149.262
C00511=1174.476,-78.974,-42.042,179.198,5.767,149.263
C00512=1174.481,-79.225,-42.031,179.196,5.767,149.264
C00513=1174.486,-79.474,-42.021,179.193,5.766,149.264
C00514=1174.492,-79.724,-42.011,179.191,5.767,149.265
C00515=1174.497,-79.974,-42.000,179.189,5.766,149.265
C00516=1174.502,-80.224,-41.990,179.187,5.766,149.266
C00517=1174.507,-80.474,-41.979,179.185,5.765,149.267
C00518=1174.512,-80.722,-41.969,179.182,5.765,149.267
C00519=1174.518,-80.972,-41.959,179.181,5.765,149.268
C00520=1174.523,-81.222,-41.948,179.178,5.765,149.269
C00521=1174.528,-81.472,-41.938,179.176,5.764,149.269
C00522=1174.534,-81.721,-41.928,179.174,5.764,149.270
C00523=1174.539,-81.972,-41.917,179.171,5.764,149.270
C00524=1174.544,-82.221,-41.907,179.169,5.763,149.271
C00525=1174.549,-82.470,-41.897,179.167,5.763,149.271
C00526=1174.554,-82.721,-41.887,179.164,5.763,149.272
C00527=1174.560,-82.970,-41.877,179.162,5.763,149.273
C00528=1174.565,-83.220,-41.866,179.160,5.762,149.273
C00529=1174.570,-83.470,-41.856,179.157,5.762,149.274
C00530=1174.576,-83.719,-41.846,179.156,5.762,149.274
C00531=1174.581,-83.969,-41.836,179.153,5.762,149.275
C00532=1174.586,-84.219,-41.825,179.151,5.761,149.276
C00533=1174.592,-84.469,-41.816,179.149,5.761,149.276
C00534=1174.597,-84.719,-41.806,179.147,5.760,149.277
C00535=1174.602,-84.969,-41.795,179.144,5.760,149.278
C00536=1174.607,-85.218,-41.786,179.143,5.760,149.278
C00537=1174.613,-85.468,-41.775,179.140,5.760,149.279
C00538=1174.618,-85.718,-41.765,179.138,5.760,149.279
C00539=1174.623,-85.967,-41.755,179.136,5.759,149.280
C00540=1174.628,-86.217,-41.745,179.133,5.759,149.281
C00541=1174.634,-86.466,-41.735,179.131,5.759,149.281
C00542=1174.639,-86.716,-41.724,179.129,5.758,149.282
C00543=1174.644,-86.966,-41.714,179.127,5.758,149.282
C00544=1174.650,-87.216,-41.705,179.124,5.758,149.283
C00545=1174.655,-87.466,-41.694,179.122,5.757,149.284
C00546=1174.660,-87.716,-41.684,179.120,5.758,149.284
C00547=1174.666,-87.965,-41.674,179.118,5.757,149.285
C00548=1174.671,-88.214,-41.664,179.115,5.756,149.285
C00549=1174.676,-88.465,-41.654,179.114,5.756,149.286
C00550=1174.681,-88.714,-41.644,179.111,5.756,149.287
C00551=1174.686,-88.964,-41.635,179.109,5.756,149.287
C00552=1174.691,-89.214,-41.624,179.107,5.756,149.288
C00553=1174.697,-89.464,-41.614,179.104,5.755,149.288
C00554=1174.703,-89.713,-41.604,179.102,5.755,149.289
C00555=1174.707,-89.963,-41.594,179.100,5.755,149.290
C00556=1174.713,-90.213,-41.585,179.098,5.755,149.290
C00557=1174.718,-90.463,-41.574,179.096,5.754,149.291
C00558=1174.723,-90.712,-41.564,179.093,5.754,149.291
C00559=1174.729,-90.962,-41.554,179.092,5.754,149.292
C00560=1174.735,-91.212,-41.545,179.089,5.753,149.293
C00561=1174.739,-91.462,-41.535,179.087,5.753,149.293
C00562=1174.745,-91.711,-41.525,179.085,5.753,149.294
C00563=1174.750,-91.961,-41.514,179.083,5.752,149.294
C00564=1174.755,-92.211,-41.505,179.080,5.753,149.295
C00565=1174.760,-92.461,-41.495,179.078,5.752,149.295
C00566=1174.765,-92.710,-41.485,179.076,5.752,149.296
C00567=1174.771,-92.960,-41.475,179.074,5.751,149.297
C00568=1174.777,-93.210,-41.466,179.071,5.751,149.297
C00569=1174.782,-93.459,-41.456,179.070,5.751,149.298
C00570=1174.787,-93.709,-41.445,179.067,5.751,149.299
C00571=1174.793,-93.960,-41.436,179.065,5.751,149.299
C00572=1174.797,-94.209,-41.426,179.063,5.750,149.300
C00573=1174.803,-94.458,-41.416,179.061,5.750,149.300
C00574=1174.808,-94.708,-41.407,179.059,5.750,149.301
C00575=1174.814,-94.958,-41.397,179.056,5.749,149.301
C00576=1174.819,-95.208,-41.386,179.054,5.750,149.302
C00577=1174.824,-95.458,-41.377,179.052,5.749,149.303
C00578=1174.829,-95.707,-41.367,179.049,5.748,149.303
C00579=1174.834,-95.957,-41.358,179.048,5.748,149.304
C00580=1174.840,-96.207,-41.348,179.045,5.748,149.305
C00581=1174.846,-96.456,-41.338,179.044,5.748,149.305
C00582=1174.850,-96.706,-41.328,179.041,5.748,149.306
C00583=1174.856,-96.956,-41.318,179.039,5.748,149.306
C00584=1174.861,-97.206,-41.309,179.037,5.747,149.307
C00585=1174.867,-97.456,-41.299,179.034,5.746,149.307
C00586=1174.872,-97.705,-41.290,179.032,5.747,149.308
C00587=1174.877,-97.955,-41.280,179.030,5.746,149.309
C00588=1174.882,-98.205,-41.271,179.028,5.747,149.309
C00589=1174.887,-98.455,-41.260,179.026,5.746,149.310
C00590=1174.893,-98.705,-41.251,179.024,5.746,149.311
C00591=1174.898,-98.954,-41.241,179.022,5.745,149.311
C00592=1174.903,-99.204,-41.232,179.019,5.745,149.312
C00593=1174.909,-99.454,-41.222,179.017,5.745,149.312
C00594=1174.915,-99.704,-41.212,179.015,5.745,149.313
C00595=1174.920,-99.953,-41.203,179.013,5.745,149.313
C00596=1174.925,-100.203,-41.194,179.010,5.744,149.314
C00597=1174.930,-100.452,-41.184,179.009,5.744,149.315
C00598=1174.935,-100.703,-41.174,179.006,5.744,149.315
C00599=1174.941,-100.952,-41.164,179.004,5.743,149.316
C00600=1174.946,-101.202,-41.155,179.002,5.744,149.317
C00601=1174.951,-101.452,-41.145,179.000,5.743,149.317
C00602=1174.957,-101.724,-41.135,178.998,5.743,149.318
C00603=1174.963,-101.995,-41.125,178.995,5.742,149.318
C00604=1174.969,-102.267,-41.114,178.993,5.742,149.319
C00605=1174.975,-102.539,-41.104,178.990,5.742,149.320
C00606=1174.980,-102.788,-41.094,178.988,5.742,149.320
C00607=1174.985,-103.039,-41.085,178.986,5.741,149.321
C00608=1174.990,-103.288,-41.075,178.984,5.741,149.321
C00609=1174.996,-103.538,-41.066,178.981,5.741,149.322
C00610=1175.001,-103.787,-41.056,178.980,5.741,149.323
C00611=1175.006,-104.037,-41.047,178.977,5.741,149.323
C00612=1175.012,-104.287,-41.038,178.976,5.741,149.324
C00613=1175.016,-104.537,-41.028,178.973,5.740,149.324
C00614=1175.022,-104.787,-41.018,178.971,5.739,149.325
C00615=1175.027,-105.036,-41.009,178.969,5.739,149.325
C00616=1175.032,-105.286,-41.000,178.966,5.739,149.326
C00617=1175.038,-105.536,-40.990,178.965,5.739,149.327
C00618=1175.043,-105.786,-40.981,178.962,5.739,149.327
C00619=1175.048,-106.036,-40.972,178.961,5.739,149.328
C00620=1175.054,-106.285,-40.962,178.958,5.738,149.329
C00621=1175.059,-106.535,-40.953,178.956,5.738,149.329
C00622=1175.065,-106.785,-40.943,178.954,5.738,149.330
C00623=1175.070,-107.034,-40.934,178.952,5.738,149.330
C00624=1175.075,-107.284,-40.925,178.950,5.737,149.331
C00625=1175.081,-107.534,-40.915,178.947,5.737,149.331
C00626=1175.086,-107.784,-40.906,178.946,5.737,149.332
C00627=1175.091,-108.033,-40.897,178.943,5.736,149.333
C00628=1175.097,-108.284,-40.887,178.941,5.736,149.333
C00629=1175.102,-108.533,-40.878,178.939,5.736,149.334
C00630=1175.107,-108.783,-40.869,178.937,5.736,149.334
C00631=1175.113,-109.033,-40.859,178.934,5.736,149.335
C00632=1175.118,-109.283,-40.850,178.933,5.736,149.335
C00633=1175.123,-109.532,-40.841,178.930,5.735,149.336
C00634=1175.129,-109.782,-40.831,178.928,5.735,149.337
C00635=1175.134,-110.032,-40.822,178.926,5.735,149.337
C00636=1175.139,-110.282,-40.813,178.924,5.735,149.338
C00637=1175.145,-110.531,-40.803,178.922,5.734,149.338
C00638=1175.150,-110.781,-40.794,178.919,5.734,149.339
C00639=1175.155,-111.031,-40.785,178.918,5.734,149.340
C00640=1175.160,-111.281,-40.776,178.915,5.733,149.340
C00641=1175.166,-111.530,-40.766,178.913,5.733,149.341
C00642=1175.171,-111.780,-40.757,178.911,5.733,149.341
C00643=1175.176,-112.030,-40.748,178.909,5.733,149.342
C00644=1175.181,-112.280,-40.740,178.907,5.732,149.342
C00645=1175.187,-112.530,-40.730,178.905,5.733,149.343
C00646=1175.193,-112.779,-40.721,178.903,5.732,149.344
C00647=1175.198,-113.029,-40.712,178.901,5.732,149.344
C00648=1175.203,-113.278,-40.703,178.898,5.732,149.345
C00649=1175.209,-113.529,-40.693,178.897,5.732,149.345
C00650=1175.214,-113.778,-40.685,178.894,5.731,149.346
C00651=1175.219,-114.028,-40.676,178.893,5.731,149.347
C00652=1175.224,-114.277,-40.666,178.890,5.731,149.347
C00653=1175.230,-114.528,-40.657,178.888,5.731,149.348
C00654=1175.235,-114.778,-40.648,178.886,5.730,149.348
C00655=1175.240,-115.027,-40.639,178.884,5.731,149.349
C00656=1175.245,-115.277,-40.630,178.882,5.730,149.349
C00657=1175.251,-115.527,-40.620,178.879,5.729,149.350
C00658=1175.256,-115.777,-40.611,178.877,5.729,149.351
C00659=1175.262,-116.026,-40.603,178.875,5.729,149.351
C00660=1175.267,-116.276,-40.593,178.873,5.729,149.352
C00661=1175.272,-116.525,-40.584,178.871,5.728,149.352
C00662=1175.278,-116.776,-40.575,178.869,5.729,149.353
C00663=1175.283,-117.025,-40.566,178.867,5.728,149.354
C00664=1175.289,-117.275,-40.557,178.865,5.728,149.354
C00665=1175.294,-117.525,-40.548,178.862,5.728,149.355
C00666=1175.299,-117.775,-40.539,178.861,5.728,149.355
C00667=1175.304,-118.025,-40.530,178.858,5.727,149.356
C00668=1175.310,-118.274,-40.522,178.857,5.727,149.356
C00669=1175.316,-118.524,-40.512,178.854,5.727,149.357
C00670=1175.321,-118.774,-40.504,178.852,5.727,149.358
C00671=1175.326,-119.024,-40.495,178.850,5.726,149.358
C00672=1175.331,-119.274,-40.486,178.848,5.727,149.359
C00673=1175.336,-119.524,-40.477,178.846,5.726,149.359
C00674=1175.342,-119.773,-40.468,178.844,5.726,149.360
C00675=1175.347,-120.023,-40.459,178.842,5.726,149.361
C00676=1175.352,-120.272,-40.451,178.840,5.726,149.361
C00677=1175.358,-120.523,-40.441,178.837,5.725,149.362
C00678=1175.364,-120.772,-40.432,178.836,5.725,149.362
C00679=1175.369,-121.022,-40.423,178.833,5.724,149.363
C00680=1175.374,-121.272,-40.414,178.831,5.725,149.363
C00681=1175.379,-121.522,-40.405,178.829,5.724,149.364
C00682=1175.385,-121.771,-40.397,178.828,5.724,149.364
C00683=1175.390,-122.021,-40.388,178.825,5.724,149.365
C00684=1175.395,-122.271,-40.379,178.823,5.724,149.366
C00685=1175.400,-122.521,-40.370,178.821,5.723,149.366
C00686=1175.405,-122.771,-40.361,178.819,5.723,149.367
C00687=1175.411,-123.020,-40.353,178.817,5.723,149.367
C00688=1175.416,-123.270,-40.344,178.815,5.723,149.368
C00689=1175.422,-123.520,-40.334,178.813,5.722,149.368
C00690=1175.427,-123.770,-40.325,178.811,5.722,149.369
C00691=1175.433,-124.020,-40.317,178.808,5.722,149.370
C00692=1175.438,-124.270,-40.308,178.807,5.722,149.370
C00693=1175.444,-124.519,-40.300,178.804,5.722,149.371
C00694=1175.449,-124.769,-40.291,178.802,5.722,149.371
C00695=1175.454,-125.019,-40.282,178.800,5.721,149.372
C00696=1175.459,-125.269,-40.273,178.798,5.721,149.373
C00697=1175.465,-125.518,-40.265,178.796,5.721,149.373
C00698=1175.470,-125.768,-40.256,178.794,5.721,149.374
C00699=1175.476,-126.018,-40.248,178.792,5.721,149.374
C00700=1175.481,-126.268,-40.239,178.790,5.720,149.375
C00701=1175.486,-126.518,-40.230,178.788,5.720,149.375
C00702=1175.492,-126.767,-40.221,178.786,5.720,149.376
C00703=1175.497,-127.017,-40.212,178.784,5.720,149.376
C00704=1175.502,-127.267,-40.203,178.782,5.719,149.377
C00705=1175.508,-127.517,-40.195,178.780,5.720,149.378
C00706=1175.087,-127.528,-40.236,178.776,5.723,149.379
C00707=1175.081,-127.278,-40.245,178.778,5.722,149.379
C00708=1175.076,-127.028,-40.253,178.780,5.723,149.378
C00709=1175.070,-126.778,-40.261,178.782,5.723,149.378
C00710=1175.065,-126.528,-40.270,178.785,5.723,149.377
C00711=1175.060,-126.279,-40.279,178.786,5.723,149.377
C00712=1175.055,-126.029,-40.288,178.788,5.724,149.376
C00713=1175.049,-125.780,-40.297,178.790,5.724,149.375
C00714=1175.044,-125.530,-40.305,178.793,5.725,149.375
C00715=1175.038,-125.279,-40.314,178.794,5.725,149.374
C00716=1175.033,-125.029,-40.323,178.797,5.725,149.374
C00717=1175.028,-124.779,-40.331,178.799,5.725,149.373
C00718=1175.022,-124.530,-40.340,178.801,5.726,149.373
C00719=1175.017,-124.280,-40.349,178.803,5.725,149.372
C00720=1175.012,-124.031,-40.358,178.805,5.726,149.372
C00721=1175.007,-123.781,-40.367,178.807,5.726,149.371
C00722=1175.001,-123.531,-40.376,178.809,5.726,149.370
C00723=1174.995,-123.281,-40.385,178.811,5.726,149.370
C00724=1174.990,-123.031,-40.393,178.814,5.727,149.369
C00725=1174.984,-122.781,-40.402,178.815,5.727,149.369
C00726=1174.979,-122.531,-40.411,178.817,5.727,149.368
C00727=1174.974,-122.281,-40.420,178.819,5.727,149.367
C00728=1174.968,-122.032,-40.428,178.822,5.728,149.367
C00729=1174.963,-121.782,-40.437,178.823,5.728,149.366
C00730=1174.958,-121.533,-40.446,178.826,5.728,149.366
C00731=1174.953,-121.283,-40.455,178.828,5.728,149.365
C00732=1174.948,-121.033,-40.464,178.830,5.728,149.365
C00733=1174.942,-120.783,-40.473,178.832,5.728,149.364
C00734=1174.937,-120.534,-40.481,178.834,5.729,149.364
C00735=1174.931,-120.284,-40.490,178.836,5.729,149.363
C00736=1174.926,-120.034,-40.499,178.838,5.730,149.362
C00737=1174.920,-119.784,-40.508,178.840,5.729,149.362
C00738=1174.915,-119.534,-40.517,178.843,5.730,149.361
C00739=1174.910,-119.284,-40.526,178.844,5.730,149.361
C00740=1174.905,-119.034,-40.535,178.847,5.730,149.360
C00741=1174.899,-118.785,-40.544,178.848,5.730,149.359
C00742=1174.894,-118.535,-40.553,178.851,5.731,149.359
C00743=1174.889,-118.286,-40.561,178.853,5.731,149.358
C00744=1174.883,-118.035,-40.571,178.855,5.731,149.358
C00745=1174.878,-117.786,-40.580,178.857,5.731,149.357
C00746=1174.873,-117.536,-40.589,178.859,5.732,149.357
C00747=1174.867,-117.286,-40.598,178.861,5.732,149.356
C00748=1174.862,-117.036,-40.606,178.863,5.732,149.355
C00749=1174.856,-116.787,-40.615,178.865,5.732,149.355
C00750=1174.851,-116.537,-40.625,178.868,5.732,149.354
C00751=1174.846,-116.288,-40.634,178.869,5.732,149.354
C00752=1174.841,-116.038,-40.643,178.872,5.733,149.353
C00753=1174.835,-115.788,-40.652,178.874,5.733,149.352
C00754=1174.830,-115.538,-40.661,178.876,5.733,149.352
C00755=1174.824,-115.288,-40.670,178.878,5.733,149.351
C00756=1174.819,-115.038,-40.679,178.880,5.734,149.351
C00757=1174.814,-114.788,-40.688,178.882,5.734,149.350
C00758=1174.809,-114.538,-40.697,178.884,5.734,149.350
C00759=1174.803,-114.289,-40.706,178.886,5.734,149.349
C00760=1174.797,-114.040,-40.716,178.889,5.735,149.348
C00761=1174.792,-113.790,-40.725,178.890,5.735,149.348
C00762=1174.787,-113.540,-40.734,178.892,5.735,149.347
C00763=1174.782,-113.290,-40.742,178.894,5.735,149.347
C00764=1174.776,-113.040,-40.752,178.897,5.736,149.346
C00765=1174.771,-112.790,-40.761,178.899,5.735,149.346
C00766=1174.766,-112.541,-40.770,178.901,5.736,149.345
C00767=1174.761,-112.291,-40.779,178.904,5.736,149.344
C00768=1174.755,-112.041,-40.789,178.905,5.736,149.344
C00769=1174.750,-111.791,-40.798,178.907,5.737,149.343
C00770=1174.745,-111.541,-40.807,178.909,5.737,149.343
C00771=1174.740,-111.292,-40.816,178.912,5.737,149.342
C00772=1174.734,-111.042,-40.826,178.914,5.737,149.341
C00773=1174.729,-110.792,-40.835,178.916,5.738,149.341
C00774=1174.723,-110.542,-40.844,178.918,5.737,149.340
C00775=1174.718,-110.292,-40.854,178.920,5.738,149.340
C00776=1174.713,-110.043,-40.863,178.922,5.738,149.339
C00777=1174.708,-109.793,-40.872,178.925,5.739,149.339
C00778=1174.702,-109.543,-40.880,178.926,5.739,149.338
C00779=1174.697,-109.293,-40.891,178.929,5.739,149.337
C00780=1174.692,-109.043,-40.900,178.930,5.739,149.337
C00781=1174.686,-108.794,-40.908,178.933,5.739,149.336
C00782=1174.680,-108.544,-40.918,178.935,5.740,149.336
C00783=1174.675,-108.295,-40.927,178.937,5.740,149.335
C00784=1174.670,-108.045,-40.936,178.940,5.740,149.334
C00785=1174.665,-107.794,-40.946,178.941,5.740,149.334
C00786=1174.660,-107.545,-40.956,178.944,5.741,149.333
C00787=1174.655,-107.295,-40.964,178.945,5.741,149.333
C00788=1174.649,-107.045,-40.974,178.948,5.741,149.332
C00789=1174.644,-106.796,-40.984,178.950,5.741,149.332
C00790=1174.639,-106.546,-40.992,178.952,5.741,149.331
C00791=1174.633,-106.296,-41.002,178.954,5.741,149.330
C00792=1174.628,-106.046,-41.012,178.956,5.742,149.330
C00793=1174.622,-105.796,-41.021,178.959,5.743,149.329
C00794=1174.617,-105.546,-41.030,178.960,5.743,149.329
C00795=1174.612,-105.297,-41.040,178.963,5.743,149.328
C00796=1174.606,-105.047,-41.049,178.965,5.743,149.327
C00797=1174.601,-104.798,-41.059,178.967,5.743,149.327
C00798=1174.595,-104.548,-41.068,178.969,5.743,149.326
C00799=1174.590,-104.298,-41.077,178.972,5.744,149.326
C00800=1174.585,-104.049,-41.087,178.973,5.744,149.325
C00801=1174.579,-103.798,-41.096,178.975,5.744,149.325
C00802=1174.575,-103.549,-41.106,178.978,5.745,149.324
C00803=1174.569,-103.299,-41.115,178.980,5.745,149.323
C00804=1174.563,-103.049,-41.124,178.982,5.745,149.323
C00805=1174.559,-102.800,-41.134,178.984,5.745,149.322
C00806=1174.553,-102.550,-41.143,178.987,5.746,149.321
C00807=1174.547,-102.278,-41.154,178.988,5.746,149.321
C00808=1174.542,-102.007,-41.164,178.991,5.746,149.320
C00809=1174.536,-101.734,-41.175,178.994,5.746,149.320
C00810=1174.530,-101.462,-41.185,178.996,5.747,149.319
C00811=1174.525,-101.213,-41.194,178.998,5.747,149.318
C00812=1174.520,-100.963,-41.205,179.000,5.747,149.318
C00813=1174.514,-100.713,-41.214,179.002,5.747,149.317
C00814=1174.509,-100.464,-41.224,179.004,5.748,149.317
C00815=1174.504,-100.214,-41.233,179.006,5.747,149.316
C00816=1174.498,-99.964,-41.243,179.009,5.748,149.315
C00817=1174.493,-99.714,-41.252,179.011,5.749,149.315
C00818=1174.487,-99.465,-41.262,179.013,5.749,149.314
C00819=1174.482,-99.215,-41.271,179.016,5.749,149.314
C00820=1174.477,-98.965,-41.281,179.017,5.749,149.313
C00821=1174.472,-98.715,-41.291,179.020,5.749,149.312
C00822=1174.466,-98.465,-41.301,179.021,5.749,149.312
C00823=1174.461,-98.216,-41.310,179.024,5.750,149.311
C00824=1174.456,-97.966,-41.320,179.026,5.751,149.311
C00825=1174.451,-97.717,-41.329,179.028,5.750,149.310
C00826=1174.445,-97.467,-41.339,179.031,5.751,149.310
C00827=1174.440,-97.217,-41.348,179.033,5.750,149.309
C00828=1174.435,-96.967,-41.359,179.035,5.751,149.308
C00829=1174.429,-96.717,-41.368,179.037,5.751,149.308
C00830=1174.424,-96.468,-41.378,179.039,5.752,149.307
C00831=1174.418,-96.218,-41.388,179.042,5.752,149.306
C00832=1174.413,-95.968,-41.397,179.043,5.752,149.306
C00833=1174.408,-95.719,-41.407,179.046,5.752,149.305
C00834=1174.403,-95.468,-41.417,179.048,5.752,149.305
C00835=1174.398,-95.219,-41.427,179.050,5.753,149.304
C00836=1174.392,-94.969,-41.437,179.053,5.754,149.304
C00837=1174.387,-94.719,-41.446,179.055,5.753,149.303
C00838=1174.381,-94.470,-41.456,179.057,5.754,149.302
C00839=1174.376,-94.220,-41.465,179.058,5.754,149.302
C00840=1174.371,-93.970,-41.476,179.061,5.754,149.301
C00841=1174.365,-93.720,-41.486,179.063,5.754,149.301
C00842=1174.361,-93.471,-41.495,179.065,5.755,149.300
C00843=1174.355,-93.221,-41.505,179.068,5.755,149.299
C00844=1174.350,-92.971,-41.515,179.070,5.755,149.299
C00845=1174.345,-92.721,-41.525,179.072,5.756,149.298
C00846=1174.339,-92.471,-41.535,179.074,5.755,149.298
C00847=1174.334,-92.222,-41.544,179.076,5.756,149.297
C00848=1174.329,-91.972,-41.554,179.079,5.757,149.296
C00849=1174.323,-91.723,-41.565,179.080,5.757,149.296
C00850=1174.318,-91.472,-41.574,179.083,5.757,149.295
C00851=1174.313,-91.223,-41.584,179.085,5.757,149.294
C00852=1174.307,-90.973,-41.594,179.087,5.757,149.294
C00853=1174.302,-90.724,-41.604,179.090,5.758,149.293
C00854=1174.297,-90.473,-41.614,179.092,5.758,149.293
C00855=1174.291,-90.223,-41.624,179.094,5.758,149.292
C00856=1174.287,-89.974,-41.634,179.096,5.758,149.292
C00857=1174.281,-89.725,-41.644,179.099,5.759,149.291
C00858=1174.276,-89.474,-41.654,179.101,5.759,149.290
C00859=1174.271,-89.225,-41.663,179.103,5.759,149.290
C00860=1174.265,-88.975,-41.673,179.105,5.760,149.289
C00861=1174.260,-88.725,-41.684,179.108,5.760,149.288
C00862=1174.255,-88.476,-41.694,179.109,5.760,149.288
C00863=1174.250,-88.226,-41.704,179.112,5.760,149.287
C00864=1174.244,-87.976,-41.713,179.114,5.760,149.287
C00865=1174.238,-87.726,-41.724,179.116,5.761,149.286
C00866=1174.234,-87.476,-41.734,179.118,5.762,149.286
C00867=1174.228,-87.227,-41.744,179.120,5.761,149.285
C00868=1174.223,-86.977,-41.754,179.123,5.762,149.284
C00869=1174.217,-86.728,-41.764,179.125,5.762,149.284
C00870=1174.213,-86.478,-41.774,179.127,5.762,149.283
C00871=1174.207,-86.228,-41.784,179.130,5.763,149.283
C00872=1174.201,-85.978,-41.794,179.131,5.763,149.282
C00873=1174.196,-85.728,-41.804,179.134,5.763,149.281
C00874=1174.192,-85.479,-41.814,179.136,5.764,149.281
C00875=1174.186,-85.229,-41.824,179.138,5.764,149.280
C00876=1174.181,-84.979,-41.835,179.140,5.764,149.280
C00877=1174.175,-84.729,-41.845,179.142,5.764,149.279
C00878=1174.170,-84.480,-41.855,179.145,5.764,149.278
C00879=1174.165,-84.231,-41.865,179.147,5.765,149.278
C00880=1174.160,-83.980,-41.875,179.149,5.765,149.277
C00881=1174.154,-83.731,-41.886,179.152,5.766,149.277
C00882=1174.149,-83.481,-41.896,179.154,5.766,149.276
C00883=1174.144,-83.231,-41.906,179.156,5.766,149.275
C00884=1174.139,-82.982,-41.916,179.158,5.766,149.275
C00885=1174.133,-82.732,-41.926,179.161,5.767,149.274
C00886=1174.128,-82.482,-41.937,179.163,5.767,149.273
C00887=1174.123,-82.232,-41.947,179.165,5.767,149.273
C00888=1174.118,-81.982,-41.958,179.167,5.767,149.272
C00889=1174.113,-81.733,-41.967,179.169,5.768,149.272
C00890=1174.107,-81.483,-41.977,179.172,5.768,149.271
C00891=1174.102,-81.233,-41.988,179.173,5.768,149.271
C00892=1174.097,-80.984,-41.998,179.176,5.769,149.270
C00893=1174.091,-80.734,-42.008,179.179,5.769,149.269
C00894=1174.086,-80.484,-42.019,179.180,5.769,149.269
C00895=1174.080,-80.234,-42.029,179.183,5.769,149.268
C00896=1174.075,-79.985,-42.039,179.185,5.770,149.268
C00897=1174.071,-79.735,-42.049,179.187,5.770,149.267
C00898=1174.065,-79.485,-42.060,179.190,5.771,149.266
C00899=1174.060,-79.235,-42.070,179.192,5.770,149.266
C00900=1174.054,-78.985,-42.080,179.194,5.771,149.265
C00901=1174.049,-78.736,-42.091,179.196,5.771,149.264
C00902=1174.044,-78.486,-42.101,179.198,5.771,149.264
C00903=1174.038,-78.237,-42.112,179.201,5.772,149.263
C00904=1174.033,-77.987,-42.122,179.203,5.772,149.263
C00905=1174.028,-77.737,-42.133,179.205,5.772,149.262
C00906=1174.022,-77.487,-42.143,179.208,5.773,149.261
C00907=1174.017,-77.237,-42.154,179.210,5.773,149.261
C00908=1174.012,-76.988,-42.164,179.212,5.773,149.260
C00909=1174.006,-76.738,-42.174,179.214,5.774,149.260
C00910=1174.001,-76.488,-42.185,179.217,5.774,149.259
C00911=1173.996,-76.217,-42.196,179.219,5.775,149.258
C00912=1173.990,-75.946,-42.207,179.221,5.775,149.258
C00913=1173.984,-75.675,-42.218,179.224,5.775,149.257
C00914=1173.979,-75.404,-42.231,179.226,5.775,149.256
C00915=1173.973,-75.154,-42.241,179.229,5.776,149.256
C00916=1173.968,-74.905,-42.251,179.231,5.776,149.255
C00917=1173.963,-74.655,-42.262,179.233,5.776,149.254
C00918=1173.957,-74.405,-42.272,179.236,5.777,149.254
C00919=1173.952,-74.155,-42.283,179.238,5.777,149.253
C00920=1173.947,-73.906,-42.293,179.240,5.777,149.253
C00921=1173.942,-73.656,-42.304,179.242,5.778,149.252
C00922=1173.936,-73.406,-42.314,179.244,5.778,149.252
C00923=1173.931,-73.156,-42.325,179.247,5.778,149.251
C00924=1173.926,-72.907,-42.336,179.249,5.779,149.250
C00925=1173.920,-72.657,-42.346,179.251,5.779,149.250
C00926=1173.915,-72.407,-42.356,179.254,5.779,149.249
C00927=1173.910,-72.158,-42.367,179.256,5.780,149.249
C00928=1173.905,-71.908,-42.378,179.258,5.779,149.248
C00929=1173.899,-71.658,-42.388,179.260,5.780,149.247
C00930=1173.895,-71.409,-42.399,179.263,5.781,149.247
C00931=1173.889,-71.159,-42.410,179.265,5.780,149.246
C00932=1173.884,-70.909,-42.420,179.267,5.781,149.245
C00933=1173.878,-70.660,-42.432,179.270,5.781,149.245
C00934=1173.873,-70.410,-42.442,179.271,5.781,149.244
C00935=1173.867,-70.160,-42.453,179.274,5.782,149.244
C00936=1173.863,-69.910,-42.464,179.276,5.783,149.243
C00937=1173.857,-69.661,-42.474,179.278,5.782,149.242
C00938=1173.852,-69.411,-42.485,179.281,5.783,149.242
C00939=1173.847,-69.162,-42.496,179.283,5.783,149.241
C00940=1173.842,-68.911,-42.506,179.286,5.784,149.240
C00941=1173.836,-68.662,-42.516,179.287,5.784,149.240
C00942=1173.832,-68.412,-42.528,179.290,5.784,149.239
C00943=1173.826,-68.162,-42.539,179.292,5.785,149.239
C00944=1173.821,-67.913,-42.550,179.294,5.785,149.238
C00945=1173.816,-67.663,-42.560,179.297,5.785,149.237
C00946=1173.810,-67.413,-42.570,179.299,5.786,149.237
C00947=1173.805,-67.163,-42.582,179.301,5.785,149.236
C00948=1173.800,-66.914,-42.592,179.303,5.786,149.236
C00949=1173.795,-66.664,-42.603,179.306,5.787,149.235
C00950=1173.789,-66.414,-42.614,179.308,5.787,149.235
C00951=1173.784,-66.165,-42.625,179.310,5.787,149.234
C00952=1173.778,-65.915,-42.636,179.313,5.787,149.233
C00953=1173.773,-65.665,-42.646,179.315,5.788,149.233
C00954=1173.769,-65.415,-42.657,179.317,5.788,149.232
C00955=1173.763,-65.166,-42.668,179.320,5.789,149.231
C00956=1173.758,-64.916,-42.680,179.322,5.789,149.231
C00957=1173.752,-64.666,-42.690,179.324,5.789,149.230
C00958=1173.747,-64.417,-42.701,179.326,5.790,149.230
C00959=1173.742,-64.166,-42.712,179.329,5.790,149.229
C00960=1173.737,-63.917,-42.723,179.331,5.791,149.228
C00961=1173.731,-63.667,-42.734,179.333,5.790,149.228
C00962=1173.726,-63.418,-42.745,179.336,5.791,149.227
C00963=1173.721,-63.168,-42.756,179.338,5.792,149.226
C00964=1173.716,-62.918,-42.766,179.340,5.791,149.226
C00965=1173.710,-62.669,-42.778,179.342,5.792,149.225
C00966=1173.705,-62.419,-42.789,179.345,5.792,149.225
C00967=1173.700,-62.170,-42.799,179.347,5.793,149.224
C00968=1173.695,-61.919,-42.810,179.349,5.793,149.223
C00969=1173.690,-61.670,-42.822,179.352,5.793,149.223
C00970=1173.684,-61.420,-42.832,179.354,5.794,149.222
C00971=1173.679,-61.170,-42.843,179.357,5.794,149.222
C00972=1173.675,-60.921,-42.855,179.359,5.794,149.221
C00973=1173.668,-60.671,-42.866,179.361,5.795,149.220
C00974=1173.664,-60.421,-42.877,179.364,5.795,149.220
C00975=1173.659,-60.172,-42.888,179.365,5.795,149.219
C00976=1173.653,-59.922,-42.898,179.368,5.796,149.218
C00977=1173.648,-59.672,-42.910,179.370,5.796,149.218
C00978=1173.642,-59.423,-42.920,179.373,5.797,149.217
C00979=1173.638,-59.173,-42.932,179.375,5.796,149.217
C00980=1173.632,-58.923,-42.944,179.377,5.797,149.216
C00981=1173.627,-58.674,-42.954,179.380,5.798,149.215
C00982=1173.622,-58.424,-42.965,179.382,5.799,149.215
C00983=1173.616,-58.174,-42.977,179.384,5.798,149.214
C00984=1173.612,-57.924,-42.988,179.387,5.799,149.213
C00985=1173.606,-57.675,-42.998,179.389,5.799,149.213
C00986=1173.601,-57.425,-43.010,179.392,5.800,149.212
C00987=1173.596,-57.175,-43.022,179.393,5.800,149.212
C00988=1173.590,-56.926,-43.032,179.396,5.800,149.211
C00989=1173.585,-56.676,-43.044,179.399,5.801,149.210
C00990=1173.580,-56.426,-43.055,179.400,5.801,149.210
C00991=1173.575,-56.177,-43.066,179.403,5.801,149.209
C00992=1173.569,-55.927,-43.077,179.405,5.802,149.209
C00993=1173.565,-55.677,-43.088,179.408,5.802,149.208
C00994=1173.560,-55.427,-43.100,179.410,5.802,149.207
C00995=1173.554,-55.178,-43.111,179.412,5.803,149.207
C00996=1173.549,-54.928,-43.122,179.415,5.803,149.206
C00997=1173.543,-54.678,-43.134,179.417,5.804,149.206
C00998=1173.539,-54.428,-43.145,179.419,5.804,149.205
C00999=1173.533,-54.179,-43.156,179.422,5.804,149.204
C01000=1173.528,-53.929,-43.168,179.424,5.805,149.204
C01001=1173.523,-53.679,-43.178,179.426,5.805,149.203
C01002=1173.517,-53.430,-43.190,179.429,5.806,149.203
C01003=1173.512,-53.180,-43.201,179.431,5.806,149.202
C01004=1173.507,-52.930,-43.213,179.433,5.806,149.201
C01005=1173.502,-52.681,-43.224,179.436,5.807,149.201
C01006=1173.497,-52.432,-43.235,179.438,5.807,149.200
C01007=1173.491,-52.181,-43.246,179.440,5.807,149.200
C01008=1173.486,-51.932,-43.258,179.442,5.808,149.199
C01009=1173.481,-51.682,-43.270,179.445,5.808,149.198
C01010=1173.476,-51.432,-43.281,179.447,5.809,149.198
C01011=1173.470,-51.183,-43.292,179.449,5.808,149.197
C01012=1173.466,-50.933,-43.304,179.452,5.809,149.196
C01013=1173.460,-50.683,-43.316,179.454,5.810,149.196
C01014=1173.456,-50.434,-43.327,179.457,5.810,149.195
C01015=1173.449,-50.163,-43.339,179.460,5.811,149.194
C01016=1173.444,-49.893,-43.352,179.462,5.811,149.194
C01017=1173.438,-49.622,-43.364,179.464,5.811,149.193
C01018=1173.432,-49.352,-43.377,179.467,5.811,149.193
C01019=1173.427,-49.103,-43.388,179.469,5.812,149.192
C01020=1173.422,-48.853,-43.400,179.471,5.813,149.191
C01021=1173.417,-48.603,-43.412,179.474,5.813,149.191
C01022=1173.411,-48.353,-43.422,179.477,5.813,149.190
C01023=1173.406,-48.103,-43.434,179.478,5.813,149.189
C01024=1173.401,-47.854,-43.445,179.481,5.814,149.189
C01025=1173.396,-47.604,-43.457,179.483,5.815,149.188
C01026=1173.391,-47.354,-43.468,179.486,5.815,149.188
C01027=1173.386,-47.104,-43.480,179.488,5.815,149.187
C01028=1173.380,-46.855,-43.492,179.490,5.816,149.186
C01029=1173.375,-46.605,-43.503,179.493,5.816,149.186
C01030=1173.370,-46.356,-43.516,179.495,5.817,149.185
C01031=1173.365,-46.107,-43.527,179.498,5.817,149.185
C01032=1173.360,-45.857,-43.539,179.500,5.817,149.184
C01033=1173.355,-45.607,-43.550,179.502,5.818,149.183
C01034=1173.349,-45.358,-43.561,179.505,5.818,149.183
C01035=1173.344,-45.108,-43.573,179.507,5.819,149.182
C01036=1173.339,-44.858,-43.585,179.509,5.819,149.181
C01037=1173.333,-44.608,-43.597,179.511,5.819,149.181
C01038=1173.328,-44.358,-43.608,179.514,5.820,149.180
C01039=1173.323,-44.109,-43.620,179.516,5.820,149.180
C01040=1173.318,-43.859,-43.632,179.519,5.821,149.179
C01041=1173.313,-43.609,-43.643,179.521,5.821,149.178
C01042=1173.307,-43.361,-43.655,179.523,5.821,149.178
C01043=1173.302,-43.111,-43.667,179.526,5.821,149.177
C01044=1173.297,-42.861,-43.678,179.528,5.822,149.177
C01045=1173.292,-42.611,-43.690,179.531,5.823,149.176
C01046=1173.286,-42.361,-43.702,179.533,5.824,149.175
C01047=1173.282,-42.111,-43.713,179.535,5.823,149.175
C01048=1173.276,-41.862,-43.725,179.538,5.824,149.174
C01049=1173.271,-41.612,-43.738,179.540,5.824,149.173
C01050=1173.267,-41.363,-43.749,179.542,5.825,149.173
C01051=1173.261,-41.113,-43.761,179.545,5.825,149.172
C01052=1173.256,-40.863,-43.773,179.547,5.826,149.172
C01053=1173.250,-40.613,-43.784,179.549,5.826,149.171
C01054=1173.245,-40.364,-43.796,179.552,5.826,149.170
C01055=1173.240,-40.115,-43.808,179.554,5.827,149.170
C01056=1173.234,-39.865,-43.820,179.557,5.827,149.169
C01057=1173.230,-39.615,-43.832,179.559,5.828,149.169
C01058=1173.225,-39.366,-43.844,179.561,5.828,149.168
C01059=1173.219,-39.116,-43.856,179.564,5.828,149.167
C01060=1173.214,-38.866,-43.868,179.566,5.829,149.167
C01061=1173.209,-38.616,-43.879,179.569,5.829,149.166
C01062=1173.204,-38.367,-43.892,179.571,5.830,149.166
C01063=1173.198,-38.117,-43.904,179.574,5.831,149.165
C01064=1173.193,-37.867,-43.916,179.576,5.830,149.164
C01065=1173.188,-37.617,-43.927,179.578,5.831,149.164
C01066=1173.183,-37.368,-43.939,179.580,5.832,149.163
C01067=1173.178,-37.118,-43.951,179.583,5.832,149.162
C01068=1173.172,-36.868,-43.963,179.585,5.833,149.162
C01069=1173.167,-36.619,-43.976,179.588,5.833,149.161
C01070=1173.163,-36.369,-43.987,179.590,5.833,149.161
C01071=1173.157,-36.119,-43.999,179.592,5.834,149.160
C01072=1173.152,-35.870,-44.012,179.595,5.834,149.159
C01073=1173.147,-35.620,-44.023,179.597,5.835,149.159
C01074=1173.141,-35.370,-44.035,179.600,5.835,149.158
C01075=1173.136,-35.121,-44.048,179.602,5.836,149.157
C01076=1173.131,-34.871,-44.059,179.604,5.836,149.157
C01077=1173.126,-34.622,-44.072,179.607,5.836,149.156
C01078=1173.121,-34.372,-44.084,179.609,5.837,149.155
C01079=1173.115,-34.122,-44.096,179.611,5.838,149.155
C01080=1173.110,-33.873,-44.108,179.614,5.838,149.154
C01081=1173.105,-33.623,-44.120,179.616,5.839,149.154
C01082=1173.100,-33.373,-44.133,179.619,5.839,149.153
C01083=1173.095,-33.124,-44.144,179.621,5.839,149.152
C01084=1173.090,-32.874,-44.157,179.623,5.840,149.152
C01085=1173.084,-32.624,-44.168,179.626,5.840,149.151
C01086=1173.079,-32.375,-44.180,179.629,5.841,149.151
C01087=1173.074,-32.125,-44.193,179.631,5.841,149.150
C01088=1173.068,-31.875,-44.205,179.633,5.842,149.149
C01089=1173.063,-31.626,-44.217,179.636,5.843,149.149
C01090=1173.058,-31.376,-44.229,179.638,5.842,149.148
C01091=1173.053,-31.127,-44.242,179.640,5.843,149.148
C01092=1173.048,-30.877,-44.253,179.642,5.843,149.147
C01093=1173.043,-30.628,-44.266,179.645,5.844,149.146
C01094=1173.037,-30.378,-44.278,179.648,5.844,149.146
C01095=1173.033,-30.128,-44.291,179.650,5.845,149.145
C01096=1173.028,-29.879,-44.303,179.653,5.846,149.144
C01097=1173.022,-29.629,-44.315,179.655,5.846,149.144
C01098=1173.017,-29.379,-44.328,179.657,5.846,149.143
C01099=1173.012,-29.129,-44.340,179.660,5.847,149.143
C01100=1173.007,-28.880,-44.352,179.662,5.847,149.142
C01101=1173.001,-28.630,-44.364,179.664,5.848,149.141
C01102=1172.996,-28.381,-44.377,179.667,5.848,149.141
C01103=1172.991,-28.131,-44.389,179.669,5.849,149.140
C01104=1172.986,-27.881,-44.401,179.672,5.849,149.140
C01105=1172.981,-27.631,-44.414,179.675,5.850,149.139
C01106=1172.976,-27.382,-44.426,179.676,5.850,149.138
C01107=1172.971,-27.132,-44.439,179.679,5.850,149.138
C01108=1172.965,-26.883,-44.451,179.681,5.851,149.137
C01109=1172.960,-26.633,-44.463,179.684,5.852,149.137
C01110=1172.955,-26.384,-44.476,179.686,5.852,149.136
C01111=1172.950,-26.134,-44.488,179.688,5.853,149.135
C01112=1172.945,-25.884,-44.501,179.691,5.853,149.135
C01113=1172.940,-25.634,-44.513,179.694,5.854,149.134
C01114=1172.935,-25.385,-44.526,179.696,5.855,149.134
C01115=1172.929,-25.135,-44.538,179.698,5.854,149.133
C01116=1172.924,-24.886,-44.550,179.701,5.855,149.132
C01117=1172.919,-24.636,-44.563,179.703,5.855,149.132
C01118=1172.914,-24.386,-44.575,179.706,5.856,149.131
C01119=1172.908,-24.117,-44.589,179.708,5.856,149.130
C01120=1172.903,-23.847,-44.603,179.711,5.857,149.130
C01121=1172.898,-23.576,-44.616,179.713,5.858,149.129
C01122=1172.891,-23.307,-44.630,179.716,5.858,149.128
C01123=1172.886,-23.058,-44.642,179.718,5.858,149.128
C01124=1172.882,-22.808,-44.655,179.721,5.859,149.127
C01125=1172.876,-22.558,-44.667,179.723,5.860,149.127
C01126=1172.871,-22.308,-44.680,179.726,5.860,149.126
C01127=1172.866,-22.059,-44.692,179.729,5.861,149.125
C01128=1172.861,-21.810,-44.705,179.731,5.861,149.125
C01129=1172.856,-21.559,-44.717,179.733,5.862,149.124
C01130=1172.850,-21.310,-44.730,179.736,5.863,149.124
C01131=1172.845,-21.060,-44.743,179.738,5.863,149.123
C01132=1172.840,-20.811,-44.756,179.740,5.863,149.122
C01133=1172.835,-20.562,-44.768,179.742,5.864,149.122
C01134=1172.830,-20.312,-44.781,179.745,5.864,149.121
C01135=1172.825,-20.062,-44.793,179.748,5.865,149.120
C01136=1172.819,-19.812,-44.806,179.750,5.865,149.120
C01137=1172.814,-19.563,-44.819,179.753,5.866,149.119
C01138=1172.809,-19.313,-44.832,179.755,5.866,149.118
C01139=1172.804,-19.063,-44.844,179.757,5.867,149.118
C01140=1172.799,-18.814,-44.857,179.760,5.868,149.117
C01141=1172.793,-18.564,-44.870,179.762,5.868,149.117
C01142=1172.789,-18.314,-44.883,179.765,5.869,149.116
C01143=1172.783,-18.064,-44.895,179.768,5.869,149.115
C01144=1172.778,-17.815,-44.908,179.770,5.870,149.115
C01145=1172.773,-17.566,-44.920,179.772,5.870,149.114
C01146=1172.768,-17.316,-44.934,179.775,5.870,149.114
C01147=1172.763,-17.066,-44.946,179.777,5.871,149.113
C01148=1172.757,-16.817,-44.959,179.779,5.871,149.112
C01149=1172.752,-16.568,-44.972,179.782,5.872,149.112
C01150=1172.747,-16.317,-44.985,179.784,5.873,149.111
C01151=1172.742,-16.068,-44.998,179.787,5.873,149.111
C01152=1172.737,-15.819,-45.010,179.790,5.874,149.110
C01153=1172.732,-15.569,-45.023,179.792,5.874,149.109
C01154=1172.726,-15.319,-45.036,179.794,5.875,149.109
C01155=1172.721,-15.070,-45.049,179.797,5.876,149.108
C01156=1172.717,-14.820,-45.062,179.799,5.876,149.107
C01157=1172.712,-14.570,-45.075,179.802,5.877,149.107
C01158=1172.706,-14.321,-45.088,179.804,5.877,149.106
C01159=1172.701,-14.071,-45.100,179.807,5.878,149.106
C01160=1172.696,-13.821,-45.113,179.809,5.878,149.105
C01161=1172.690,-13.572,-45.127,179.812,5.879,149.104
C01162=1172.685,-13.322,-45.139,179.814,5.880,149.104
C01163=1172.681,-13.072,-45.152,179.816,5.879,149.103
C01164=1172.675,-12.823,-45.165,179.818,5.880,149.103
C01165=1172.671,-12.573,-45.179,179.821,5.881,149.102
C01166=1172.665,-12.324,-45.192,179.823,5.881,149.101
C01167=1172.660,-12.074,-45.205,179.826,5.882,149.101
C01168=1172.655,-11.824,-45.218,179.829,5.882,149.100
C01169=1172.650,-11.575,-45.230,179.831,5.883,149.100
C01170=1172.644,-11.325,-45.244,179.833,5.884,149.099
C01171=1172.639,-11.075,-45.257,179.836,5.884,149.098
C01172=1172.634,-10.826,-45.269,179.838,5.885,149.098
C01173=1172.629,-10.577,-45.283,179.841,5.885,149.097
C01174=1172.624,-10.327,-45.296,179.844,5.886,149.096
C01175=1172.618,-10.077,-45.309,179.846,5.887,149.096
C01176=1172.614,-9.827,-45.322,179.848,5.887,149.095
C01177=1172.609,-9.578,-45.335,179.851,5.887,149.095
C01178=1172.603,-9.328,-45.348,179.853,5.888,149.094
C01179=1172.599,-9.079,-45.362,179.856,5.889,149.093
C01180=1172.593,-8.829,-45.375,179.858,5.890,149.093
C01181=1172.588,-8.579,-45.388,179.861,5.890,149.092
C01182=1172.583,-8.330,-45.400,179.863,5.890,149.092
C01183=1172.578,-8.081,-45.414,179.866,5.891,149.091
C01184=1172.573,-7.831,-45.427,179.868,5.892,149.090
C01185=1172.567,-7.581,-45.441,179.871,5.892,149.090
C01186=1172.563,-7.331,-45.453,179.873,5.893,149.089
C01187=1172.557,-7.082,-45.467,179.876,5.894,149.089
C01188=1172.553,-6.832,-45.480,179.878,5.894,149.088
C01189=1172.547,-6.583,-45.494,179.880,5.895,149.087
C01190=1172.542,-6.333,-45.507,179.883,5.895,149.087
C01191=1172.537,-6.084,-45.520,179.885,5.896,149.086
C01192=1172.532,-5.834,-45.533,179.888,5.897,149.086
C01193=1172.527,-5.584,-45.546,179.891,5.897,149.085
C01194=1172.522,-5.335,-45.560,179.893,5.898,149.084
C01195=1172.517,-5.085,-45.573,179.895,5.898,149.084
C01196=1172.511,-4.836,-45.586,179.898,5.899,149.083
C01197=1172.507,-4.586,-45.600,179.900,5.900,149.083
C01198=1172.501,-4.337,-45.613,179.903,5.900,149.082
C01199=1172.496,-4.086,-45.627,179.906,5.900,149.081
C01200=1172.491,-3.838,-45.640,179.908,5.901,149.081
C01201=1172.486,-3.587,-45.653,179.910,5.902,149.080
C01202=1172.481,-3.339,-45.667,179.913,5.903,149.080
C01203=1172.476,-3.088,-45.680,179.915,5.903,149.079
C01204=1172.471,-2.839,-45.693,179.918,5.904,149.078
C01205=1172.466,-2.589,-45.707,179.920,5.904,149.078
C01206=1172.460,-2.340,-45.720,179.923,5.905,149.077
C01207=1172.455,-2.090,-45.734,179.925,5.905,149.076
C01208=1172.450,-1.841,-45.747,179.928,5.906,149.076
C01209=1172.445,-1.591,-45.760,179.930,5.907,149.075
C01210=1172.440,-1.342,-45.774,179.933,5.907,149.074
C01211=1172.435,-1.092,-45.787,179.935,5.908,149.074
C01212=1172.429,-0.843,-45.801,179.938,5.908,149.073
C01213=1172.424,-0.592,-45.815,179.940,5.909,149.073
C01214=1172.419,-0.344,-45.828,179.943,5.910,149.072
C01215=1172.414,-0.093,-45.841,179.945,5.910,149.071
C01216=1172.409,0.155,-45.855,179.947,5.911,149.071
C01217=1172.404,0.406,-45.868,179.950,5.911,149.070
C01218=1172.398,0.655,-45.882,179.953,5.912,149.070
C01219=1172.394,0.905,-45.895,179.955,5.913,149.069
C01220=1172.389,1.155,-45.909,179.957,5.913,149.068
C01221=1172.383,1.404,-45.923,179.960,5.914,149.068
C01222=1172.379,1.654,-45.936,179.962,5.914,149.067
C01223=1172.373,1.922,-45.951,179.965,5.915,149.067
C01224=1172.367,2.192,-45.966,179.968,5.916,149.066
C01225=1172.362,2.461,-45.981,179.971,5.917,149.065
C01226=1172.356,2.731,-45.995,179.973,5.917,149.065
C01227=1172.351,2.980,-46.009,179.976,5.918,149.064
C01228=1172.347,3.230,-46.023,179.978,5.918,149.063
C01229=1172.341,3.479,-46.036,179.980,5.919,149.063
C01230=1172.336,3.729,-46.050,179.983,5.920,149.062
C01231=1172.331,3.978,-46.064,179.986,5.920,149.062
C01232=1172.326,4.228,-46.077,179.988,5.921,149.061
C01233=1172.321,4.478,-46.091,179.991,5.921,149.060
C01234=1172.316,4.727,-46.104,179.993,5.922,149.060
C01235=1172.311,4.977,-46.118,179.995,5.923,149.059
C01236=1172.306,5.226,-46.133,179.999,5.924,149.059
C01237=1172.300,5.475,-46.147,-179.999,5.925,149.058
C01238=1172.296,5.725,-46.159,-179.996,5.925,149.057
C01239=1172.291,5.975,-46.174,-179.994,5.926,149.057
C01240=1172.285,6.224,-46.188,-179.992,5.927,149.056
C01241=1172.280,6.474,-46.201,-179.989,5.927,149.056
C01242=1172.276,6.724,-46.215,-179.986,5.928,149.055
C01243=1172.270,6.973,-46.229,-179.984,5.928,149.054
C01244=1172.265,7.223,-46.243,-179.982,5.929,149.054
C01245=1172.260,7.473,-46.257,-179.979,5.930,149.053
C01246=1172.254,7.722,-46.271,-179.977,5.930,149.053
C01247=1172.250,7.971,-46.284,-179.974,5.931,149.052
C01248=1172.245,8.221,-46.299,-179.972,5.932,149.052
C01249=1172.239,8.471,-46.312,-179.969,5.932,149.051
C01250=1172.234,8.720,-46.326,-179.967,5.932,149.050
C01251=1172.229,8.970,-46.340,-179.964,5.934,149.050
C01252=1172.224,9.219,-46.354,-179.961,5.935,149.049
C01253=1172.220,9.468,-46.368,-179.959,5.935,149.049
C01254=1172.214,9.719,-46.381,-179.956,5.936,149.048
C01255=1172.209,9.968,-46.395,-179.954,5.936,149.047
C01256=1172.204,10.217,-46.410,-179.952,5.937,149.047
C01257=1172.199,10.467,-46.424,-179.949,5.938,149.046
C01258=1172.193,10.716,-46.438,-179.946,5.938,149.045
C01259=1172.188,10.966,-46.452,-179.944,5.939,149.045
C01260=1172.183,11.216,-46.466,-179.941,5.939,149.044
C01261=1172.179,11.466,-46.479,-179.939,5.940,149.044
C01262=1172.173,11.715,-46.493,-179.937,5.941,149.043
C01263=1172.168,11.964,-46.508,-179.933,5.942,149.042
C01264=1172.163,12.214,-46.522,-179.931,5.943,149.042
C01265=1172.158,12.464,-46.536,-179.929,5.943,149.041
C01266=1172.153,12.713,-46.550,-179.926,5.944,149.041
C01267=1172.148,12.963,-46.564,-179.924,5.945,149.040
C01268=1172.143,13.212,-46.579,-179.921,5.945,149.039
C01269=1172.138,13.462,-46.593,-179.919,5.946,149.039
C01270=1172.132,13.711,-46.607,-179.916,5.946,149.038
C01271=1172.127,13.961,-46.621,-179.914,5.947,149.038
C01272=1172.123,14.210,-46.635,-179.911,5.948,149.037
C01273=1172.118,14.460,-46.650,-179.908,5.949,149.036
C01274=1172.112,14.709,-46.663,-179.906,5.950,149.036
C01275=1172.107,14.959,-46.678,-179.903,5.950,149.035
C01276=1172.102,15.209,-46.692,-179.901,5.951,149.035
C01277=1172.097,15.458,-46.706,-179.899,5.952,149.034
C01278=1172.092,15.707,-46.720,-179.896,5.952,149.033
C01279=1172.087,15.957,-46.734,-179.894,5.953,149.033
C01280=1172.082,16.207,-46.749,-179.891,5.953,149.032
C01281=1172.077,16.456,-46.763,-179.888,5.954,149.032
C01282=1172.072,16.706,-46.777,-179.886,5.956,149.031
C01283=1172.066,16.955,-46.791,-179.883,5.956,149.031
C01284=1172.061,17.205,-46.806,-179.880,5.957,149.030
C01285=1172.056,17.454,-46.820,-179.878,5.957,149.029
C01286=1172.051,17.704,-46.834,-179.876,5.958,149.029
C01287=1172.046,17.954,-46.848,-179.873,5.959,149.028
C01288=1172.042,18.203,-46.863,-179.871,5.959,149.028
C01289=1172.036,18.452,-46.877,-179.868,5.960,149.027
C01290=1172.031,18.702,-46.892,-179.865,5.961,149.026
C01291=1172.026,18.951,-46.906,-179.863,5.962,149.026
C01292=1172.021,19.201,-46.920,-179.861,5.963,149.025
C01293=1172.016,19.451,-46.934,-179.858,5.963,149.025
C01294=1172.011,19.701,-46.949,-179.855,5.964,149.024
C01295=1172.006,19.950,-46.964,-179.853,5.964,149.023
C01296=1172.000,20.199,-46.978,-179.850,5.965,149.023
C01297=1171.996,20.449,-46.992,-179.848,5.967,149.022
C01298=1171.991,20.698,-47.007,-179.845,5.967,149.022
C01299=1171.986,20.948,-47.021,-179.842,5.968,149.021
C01300=1171.981,21.197,-47.036,-179.840,5.968,149.021
C01301=1171.976,21.447,-47.050,-179.838,5.969,149.020
C01302=1171.971,21.697,-47.065,-179.835,5.970,149.019
C01303=1171.965,21.947,-47.079,-179.833,5.970,149.019
C01304=1171.960,22.195,-47.094,-179.830,5.971,149.018
C01305=1171.955,22.445,-47.108,-179.827,5.972,149.018
C01306=1171.950,22.694,-47.123,-179.825,5.973,149.017
C01307=1171.945,22.944,-47.137,-179.822,5.973,149.016
C01308=1171.941,23.193,-47.152,-179.820,5.974,149.016
C01309=1171.935,23.443,-47.167,-179.817,5.975,149.015
C01310=1171.930,23.693,-47.181,-179.815,5.975,149.015
C01311=1171.925,23.942,-47.196,-179.812,5.977,149.014
C01312=1171.920,24.192,-47.210,-179.809,5.977,149.013
C01313=1171.915,24.442,-47.225,-179.807,5.978,149.013
C01314=1171.910,24.691,-47.240,-179.804,5.979,149.012
C01315=1171.905,24.941,-47.254,-179.802,5.979,149.012
C01316=1171.899,25.190,-47.268,-179.800,5.980,149.011
C01317=1171.895,25.439,-47.283,-179.796,5.981,149.010
C01318=1171.889,25.689,-47.298,-179.794,5.982,149.010
C01319=1171.884,25.938,-47.312,-179.792,5.983,149.009
C01320=1171.880,26.188,-47.327,-179.789,5.983,149.009
C01321=1171.875,26.437,-47.342,-179.787,5.984,149.008
C01322=1171.869,26.687,-47.357,-179.784,5.986,149.008
C01323=1171.864,26.936,-47.372,-179.781,5.986,149.007
C01324=1171.860,27.185,-47.387,-179.779,5.986,149.006
C01325=1171.855,27.435,-47.401,-179.777,5.987,149.006
C01326=1171.849,27.685,-47.416,-179.774,5.988,149.005
C01327=1171.844,27.954,-47.431,-179.771,5.989,149.004
C01328=1171.839,28.223,-47.447,-179.768,5.990,149.004
C01329=1171.833,28.492,-47.463,-179.766,5.990,149.003
C01330=1171.828,28.760,-47.480,-179.763,5.992,149.003
C01331=1171.822,29.010,-47.495,-179.760,5.992,149.002
C01332=1171.818,29.259,-47.510,-179.758,5.993,149.002
C01333=1171.813,29.509,-47.524,-179.755,5.994,149.001
C01334=1171.807,29.758,-47.540,-179.753,5.994,149.000
C01335=1171.802,30.008,-47.554,-179.750,5.996,149.000
C01336=1171.798,30.257,-47.569,-179.747,5.996,148.999
C01337=1171.792,30.507,-47.584,-179.745,5.997,148.999
C01338=1171.787,30.756,-47.599,-179.742,5.998,148.998
C01339=1171.782,31.006,-47.613,-179.740,5.998,148.997
C01340=1171.777,31.255,-47.629,-179.737,6.000,148.997
C01341=1171.772,31.505,-47.643,-179.734,6.000,148.996
C01342=1171.767,31.754,-47.658,-179.732,6.001,148.996
C01343=1171.762,32.003,-47.673,-179.729,6.001,148.995
C01344=1171.757,32.253,-47.688,-179.727,6.002,148.995
C01345=1171.752,32.503,-47.703,-179.724,6.004,148.994
C01346=1171.747,32.752,-47.718,-179.722,6.004,148.993
C01347=1171.742,33.002,-47.734,-179.719,6.005,148.993
C01348=1171.737,33.252,-47.749,-179.717,6.005,148.992
C01349=1171.732,33.501,-47.763,-179.714,6.007,148.992
C01350=1171.727,33.751,-47.778,-179.711,6.008,148.991
C01351=1171.722,34.000,-47.793,-179.709,6.008,148.990
C01352=1171.717,34.250,-47.808,-179.706,6.009,148.990
C01353=1171.712,34.499,-47.823,-179.704,6.010,148.989
C01354=1171.707,34.748,-47.839,-179.701,6.011,148.989
C01355=1171.702,34.997,-47.854,-179.698,6.012,148.988
C01356=1171.696,35.247,-47.869,-179.696,6.012,148.988
C01357=1171.692,35.496,-47.884,-179.694,6.013,148.987
C01358=1171.687,35.747,-47.900,-179.691,6.015,148.986
C01359=1171.682,35.996,-47.914,-179.688,6.015,148.986
C01360=1171.676,36.246,-47.930,-179.686,6.016,148.985
C01361=1171.672,36.495,-47.945,-179.683,6.016,148.985
C01362=1171.666,36.744,-47.960,-179.680,6.018,148.984
C01363=1171.661,36.994,-47.974,-179.678,6.019,148.984
C01364=1171.656,37.243,-47.990,-179.675,6.019,148.983
C01365=1171.651,37.492,-48.005,-179.673,6.020,148.982
C01366=1171.647,37.742,-48.021,-179.671,6.020,148.982
C01367=1171.642,37.992,-48.036,-179.667,6.022,148.981
C01368=1171.636,38.242,-48.051,-179.665,6.023,148.981
C01369=1171.631,38.491,-48.066,-179.663,6.023,148.980
C01370=1171.626,38.740,-48.081,-179.660,6.024,148.979
C01371=1171.621,38.989,-48.097,-179.657,6.025,148.979
C01372=1171.617,39.239,-48.112,-179.655,6.026,148.978
C01373=1171.611,39.489,-48.128,-179.652,6.027,148.978
C01374=1171.607,39.738,-48.143,-179.650,6.027,148.977
C01375=1171.601,39.988,-48.158,-179.647,6.029,148.977
C01376=1171.596,40.237,-48.173,-179.644,6.029,148.976
C01377=1171.592,40.487,-48.189,-179.642,6.030,148.975
C01378=1171.586,40.736,-48.204,-179.640,6.031,148.975
C01379=1171.581,40.986,-48.220,-179.637,6.032,148.974
C01380=1171.576,41.235,-48.235,-179.634,6.033,148.974
C01381=1171.571,41.484,-48.250,-179.632,6.034,148.973
C01382=1171.567,41.734,-48.266,-179.629,6.035,148.973
C01383=1171.561,41.983,-48.281,-179.626,6.035,148.972
C01384=1171.556,42.233,-48.297,-179.624,6.036,148.971
C01385=1171.551,42.482,-48.312,-179.621,6.037,148.971
C01386=1171.546,42.731,-48.328,-179.619,6.038,148.970
C01387=1171.541,42.981,-48.344,-179.616,6.039,148.970
C01388=1171.537,43.231,-48.359,-179.614,6.040,148.969
C01389=1171.531,43.480,-48.374,-179.611,6.040,148.969
C01390=1171.526,43.729,-48.390,-179.608,6.042,148.968
C01391=1171.521,43.979,-48.406,-179.606,6.043,148.967
C01392=1171.516,44.229,-48.421,-179.603,6.043,148.967
C01393=1171.511,44.478,-48.436,-179.600,6.045,148.966
C01394=1171.506,44.727,-48.452,-179.598,6.045,148.966
C01395=1171.502,44.977,-48.467,-179.596,6.046,148.965
C01396=1171.496,45.227,-48.483,-179.593,6.047,148.964
C01397=1171.491,45.476,-48.498,-179.590,6.048,148.964
C01398=1171.486,45.726,-48.514,-179.588,6.049,148.963
C01399=1171.481,45.975,-48.529,-179.585,6.050,148.963
C01400=1171.476,46.224,-48.546,-179.582,6.051,148.962
C01401=1171.471,46.473,-48.561,-179.580,6.052,148.962
C01402=1171.466,46.723,-48.577,-179.577,6.052,148.961
C01403=1171.461,46.973,-48.592,-179.574,6.054,148.960
C01404=1171.456,47.222,-48.608,-179.572,6.054,148.960
C01405=1171.451,47.472,-48.624,-179.569,6.055,148.959
C01406=1171.446,47.721,-48.639,-179.567,6.056,148.959
C01407=1171.441,47.970,-48.656,-179.564,6.057,148.958
C01408=1171.437,48.220,-48.671,-179.562,6.058,148.958
C01409=1171.431,48.469,-48.687,-179.559,6.058,148.957
C01410=1171.426,48.719,-48.702,-179.556,6.060,148.957
C01411=1171.421,48.969,-48.718,-179.554,6.061,148.956
C01412=1171.416,49.218,-48.734,-179.552,6.062,148.956
C01413=1171.411,49.467,-48.749,-179.548,6.063,148.955
C01414=1171.407,49.717,-48.765,-179.546,6.063,148.954
C01415=1171.401,49.966,-48.781,-179.544,6.064,148.954
C01416=1171.396,50.215,-48.797,-179.540,6.065,148.953
C01417=1171.391,50.465,-48.813,-179.538,6.066,148.953
C01418=1171.386,50.715,-48.829,-179.536,6.067,148.952
C01419=1171.381,50.964,-48.844,-179.533,6.069,148.952
C01420=1171.377,51.213,-48.860,-179.530,6.069,148.951
C01421=1171.372,51.463,-48.876,-179.528,6.070,148.950
C01422=1171.367,51.713,-48.892,-179.525,6.071,148.950
C01423=1171.362,51.961,-48.908,-179.523,6.072,148.949
C01424=1171.356,52.211,-48.924,-179.520,6.073,148.949
C01425=1171.351,52.461,-48.940,-179.518,6.073,148.948
C01426=1171.346,52.710,-48.956,-179.515,6.075,148.948
C01427=1171.342,52.960,-48.972,-179.513,6.076,148.947
C01428=1171.336,53.209,-48.988,-179.509,6.077,148.947
C01429=1171.331,53.458,-49.004,-179.507,6.077,148.946
C01430=1171.326,53.708,-49.020,-179.504,6.078,148.945
C01431=1171.321,53.977,-49.037,-179.501,6.080,148.945
C01432=1171.316,54.244,-49.055,-179.499,6.081,148.944
C01433=1171.311,54.514,-49.072,-179.496,6.082,148.944
C01434=1171.305,54.782,-49.089,-179.493,6.082,148.943
C01435=1171.300,55.032,-49.105,-179.491,6.084,148.943
C01436=1171.295,55.281,-49.121,-179.488,6.085,148.942
C01437=1171.290,55.530,-49.137,-179.486,6.085,148.941
C01438=1171.285,55.780,-49.154,-179.483,6.087,148.941
C01439=1171.280,56.029,-49.169,-179.480,6.088,148.940
C01440=1171.275,56.279,-49.186,-179.478,6.088,148.940
C01441=1171.270,56.528,-49.201,-179.474,6.089,148.939
C01442=1171.265,56.777,-49.218,-179.472,6.090,148.939
C01443=1171.260,57.027,-49.234,-179.470,6.091,148.938
C01444=1171.255,57.276,-49.250,-179.467,6.092,148.937
C01445=1171.250,57.526,-49.266,-179.464,6.093,148.937
C01446=1171.245,57.775,-49.282,-179.462,6.095,148.936
C01447=1171.240,58.025,-49.298,-179.459,6.095,148.936
C01448=1171.235,58.274,-49.314,-179.457,6.096,148.935
C01449=1171.231,58.524,-49.330,-179.454,6.097,148.935
C01450=1171.225,58.773,-49.347,-179.451,6.098,148.934
C01451=1171.221,59.022,-49.363,-179.449,6.099,148.933
C01452=1171.215,59.272,-49.380,-179.446,6.100,148.933
C01453=1171.210,59.521,-49.396,-179.443,6.101,148.932
C01454=1171.205,59.771,-49.412,-179.441,6.103,148.932
C01455=1171.201,60.020,-49.429,-179.438,6.103,148.931
C01456=1171.195,60.269,-49.445,-179.436,6.104,148.931
C01457=1171.191,60.519,-49.461,-179.433,6.105,148.930
C01458=1171.186,60.768,-49.477,-179.431,6.106,148.930
C01459=1171.181,61.017,-49.494,-179.428,6.107,148.929
C01460=1171.176,61.268,-49.510,-179.425,6.108,148.929
C01461=1171.171,61.516,-49.527,-179.423,6.109,148.928
C01462=1171.166,61.766,-49.543,-179.420,6.111,148.928
C01463=1171.161,62.015,-49.559,-179.417,6.111,148.927
C01464=1171.156,62.265,-49.576,-179.415,6.112,148.926
C01465=1171.151,62.514,-49.592,-179.412,6.113,148.926
C01466=1171.146,62.763,-49.609,-179.410,6.114,148.925
C01467=1171.141,63.014,-49.625,-179.406,6.115,148.925
C01468=1171.136,63.262,-49.641,-179.404,6.116,148.924
C01469=1171.132,63.512,-49.658,-179.402,6.117,148.924
C01470=1171.126,63.761,-49.674,-179.399,6.119,148.923
C01471=1171.121,64.011,-49.691,-179.396,6.119,148.922
C01472=1171.116,64.260,-49.708,-179.394,6.121,148.922
C01473=1171.111,64.509,-49.724,-179.391,6.121,148.921
C01474=1171.107,64.759,-49.741,-179.389,6.122,148.921
C01475=1171.101,65.008,-49.756,-179.386,6.123,148.920
C01476=1171.096,65.258,-49.773,-179.383,6.124,148.920
C01477=1171.092,65.507,-49.790,-179.381,6.126,148.919
C01478=1171.087,65.756,-49.806,-179.378,6.127,148.919
C01479=1171.082,66.006,-49.823,-179.375,6.128,148.918
C01480=1171.076,66.255,-49.840,-179.373,6.129,148.918
C01481=1171.072,66.504,-49.857,-179.371,6.130,148.917
C01482=1171.067,66.754,-49.873,-179.367,6.131,148.917
C01483=1171.061,67.003,-49.889,-179.365,6.132,148.916
C01484=1171.057,67.253,-49.906,-179.362,6.133,148.915
C01485=1171.052,67.502,-49.923,-179.360,6.134,148.915
C01486=1171.047,67.751,-49.939,-179.357,6.135,148.914
C01487=1171.042,68.001,-49.956,-179.354,6.136,148.914
C01488=1171.038,68.250,-49.973,-179.352,6.137,148.913
C01489=1171.033,68.499,-49.989,-179.349,6.138,148.913
C01490=1171.027,68.749,-50.007,-179.346,6.139,148.912
C01491=1171.023,68.999,-50.023,-179.344,6.141,148.912
C01492=1171.018,69.247,-50.040,-179.341,6.141,148.911
C01493=1171.013,69.497,-50.057,-179.338,6.143,148.911
C01494=1171.008,69.747,-50.073,-179.336,6.143,148.910
C01495=1171.003,69.996,-50.091,-179.334,6.144,148.910
C01496=1170.998,70.245,-50.107,-179.330,6.146,148.909
C01497=1170.993,70.495,-50.124,-179.328,6.146,148.909
C01498=1170.988,70.744,-50.141,-179.325,6.148,148.908
C01499=1170.983,70.993,-50.157,-179.323,6.149,148.907
C01500=1170.978,71.243,-50.175,-179.320,6.150,148.907
C01501=1170.973,71.493,-50.191,-179.317,6.151,148.906
C01502=1170.969,71.742,-50.208,-179.315,6.153,148.906
C01503=1170.963,71.991,-50.225,-179.312,6.153,148.905
C01504=1170.958,72.241,-50.241,-179.309,6.155,148.905
C01505=1170.953,72.490,-50.259,-179.307,6.155,148.904
C01506=1170.948,72.739,-50.275,-179.305,6.156,148.904
C01507=1170.943,72.988,-50.293,-179.301,6.158,148.903
C01508=1170.939,73.238,-50.310,-179.299,6.158,148.903
C01509=1170.934,73.488,-50.327,-179.296,6.160,148.902
C01510=1170.929,73.737,-50.344,-179.294,6.161,148.902
C01511=1170.923,73.986,-50.361,-179.291,6.162,148.901
C01512=1170.919,74.236,-50.377,-179.288,6.163,148.900
C01513=1170.914,74.485,-50.394,-179.286,6.165,148.900
C01514=1170.909,74.734,-50.412,-179.283,6.165,148.899
C01515=1170.904,74.983,-50.428,-179.280,6.167,148.899
C01516=1170.899,75.233,-50.445,-179.278,6.167,148.898
C01517=1170.894,75.483,-50.463,-179.275,6.169,148.898
C01518=1170.889,75.732,-50.479,-179.273,6.170,148.897
C01519=1170.884,75.981,-50.497,-179.270,6.171,148.897
C01520=1170.879,76.230,-50.514,-179.268,6.172,148.896
C01521=1170.874,76.480,-50.531,-179.264,6.173,148.896
C01522=1170.870,76.729,-50.548,-179.262,6.174,148.895
C01523=1170.865,76.979,-50.566,-179.259,6.176,148.895
C01524=1170.860,77.228,-50.582,-179.257,6.176,148.894
C01525=1170.854,77.477,-50.599,-179.254,6.178,148.894
C01526=1170.850,77.726,-50.617,-179.251,6.179,148.893
C01527=1170.845,77.976,-50.634,-179.249,6.180,148.893
C01528=1170.840,78.226,-50.651,-179.246,6.181,148.892
C01529=1170.836,78.475,-50.668,-179.243,6.183,148.892
C01530=1170.830,78.724,-50.686,-179.241,6.183,148.891
C01531=1170.825,78.974,-50.703,-179.238,6.185,148.891
C01532=1170.821,79.222,-50.720,-179.235,6.185,148.890
C01533=1170.815,79.472,-50.737,-179.233,6.187,148.889
C01534=1170.811,79.722,-50.754,-179.231,6.188,148.889
C01535=1170.806,79.990,-50.773,-179.227,6.189,148.888
C01536=1170.800,80.258,-50.792,-179.225,6.190,148.888
C01537=1170.794,80.527,-50.810,-179.222,6.192,148.887
C01538=1170.790,80.795,-50.828,-179.219,6.193,148.887
C01539=1170.785,81.045,-50.846,-179.217,6.194,148.886
C01540=1170.780,81.294,-50.864,-179.213,6.195,148.886
C01541=1170.775,81.543,-50.881,-179.211,6.196,148.885
C01542=1170.770,81.792,-50.898,-179.208,6.197,148.884
C01543=1170.765,82.041,-50.916,-179.205,6.199,148.884
C01544=1170.759,82.291,-50.933,-179.203,6.200,148.884
C01545=1170.755,82.540,-50.951,-179.200,6.201,148.883
C01546=1170.750,82.790,-50.968,-179.198,6.202,148.883
C01547=1170.745,83.039,-50.986,-179.195,6.203,148.882
C01548=1170.741,83.289,-51.002,-179.192,6.204,148.881
C01549=1170.736,83.538,-51.020,-179.190,6.206,148.881
C01550=1170.731,83.788,-51.038,-179.187,6.207,148.880
C01551=1170.726,84.037,-51.056,-179.184,6.208,148.880
C01552=1170.721,84.286,-51.072,-179.182,6.209,148.879
C01553=1170.716,84.535,-51.090,-179.179,6.210,148.879
C01554=1170.711,84.785,-51.108,-179.177,6.211,148.878
C01555=1170.706,85.034,-51.126,-179.174,6.213,148.878
C01556=1170.702,85.283,-51.143,-179.172,6.214,148.877
C01557=1170.697,85.533,-51.160,-179.168,6.215,148.877
C01558=1170.692,85.782,-51.178,-179.166,6.217,148.876
C01559=1170.687,86.031,-51.196,-179.163,6.217,148.876
C01560=1170.681,86.280,-51.213,-179.160,6.219,148.875
C01561=1170.676,86.530,-51.231,-179.158,6.220,148.875
C01562=1170.672,86.779,-51.248,-179.155,6.221,148.874
C01563=1170.667,87.028,-51.266,-179.153,6.222,148.874
C01564=1170.662,87.277,-51.284,-179.150,6.224,148.873
C01565=1170.657,87.527,-51.301,-179.147,6.224,148.873
C01566=1170.652,87.776,-51.319,-179.145,6.226,148.872
C01567=1170.647,88.026,-51.337,-179.141,6.227,148.872
C01568=1170.643,88.275,-51.355,-179.139,6.228,148.871
C01569=1170.638,88.525,-51.372,-179.137,6.230,148.871
C01570=1170.633,88.774,-51.390,-179.134,6.230,148.870
C01571=1170.628,89.023,-51.408,-179.131,6.232,148.870
C01572=1170.623,89.273,-51.426,-179.129,6.233,148.869
C01573=1170.618,89.522,-51.443,-179.126,6.234,148.869
C01574=1170.613,89.772,-51.461,-179.123,6.236,148.868
C01575=1170.608,90.021,-51.479,-179.121,6.237,148.868
C01576=1170.603,90.270,-51.497,-179.118,6.238,148.867
C01577=1170.598,90.520,-51.514,-179.116,6.239,148.867
C01578=1170.593,90.769,-51.532,-179.113,6.241,148.866
C01579=1170.589,91.018,-51.550,-179.110,6.241,148.866
C01580=1170.584,91.267,-51.568,-179.107,6.243,148.865
C01581=1170.579,91.516,-51.586,-179.104,6.245,148.865
C01582=1170.574,91.765,-51.604,-179.102,6.245,148.864
C01583=1170.569,92.014,-51.622,-179.099,6.247,148.864
C01584=1170.564,92.264,-51.639,-179.097,6.248,148.863
C01585=1170.560,92.514,-51.657,-179.094,6.249,148.863
C01586=1170.555,92.763,-51.675,-179.091,6.251,148.862
C01587=1170.550,93.012,-51.693,-179.089,6.252,148.862
C01588=1170.545,93.262,-51.711,-179.086,6.253,148.861
C01589=1170.540,93.511,-51.729,-179.084,6.254,148.861
C01590=1170.535,93.760,-51.747,-179.081,6.256,148.860
C01591=1170.530,94.009,-51.765,-179.078,6.257,148.860
C01592=1170.525,94.258,-51.783,-179.075,6.258,148.859
C01593=1170.521,94.507,-51.801,-179.073,6.259,148.859
C01594=1170.516,94.757,-51.819,-179.070,6.260,148.858
C01595=1170.511,95.007,-51.837,-179.067,6.262,148.858
C01596=1170.506,95.256,-51.856,-179.065,6.263,148.857
C01597=1170.501,95.505,-51.874,-179.062,6.264,148.857
C01598=1170.496,95.754,-51.892,-179.059,6.266,148.856
C01599=1170.491,96.004,-51.910,-179.057,6.266,148.856
C01600=1170.486,96.253,-51.928,-179.054,6.268,148.855
C01601=1170.482,96.503,-51.946,-179.051,6.270,148.855
C01602=1170.477,96.752,-51.964,-179.049,6.270,148.854
C01603=1170.472,97.001,-51.982,-179.046,6.272,148.854
C01604=1170.467,97.250,-52.000,-179.043,6.274,148.853
C01605=1170.462,97.499,-52.018,-179.041,6.274,148.853
C01606=1170.457,97.749,-52.037,-179.038,6.276,148.852
C01607=1170.452,97.999,-52.055,-179.036,6.277,148.852
C01608=1170.447,98.248,-52.073,-179.033,6.278,148.851
C01609=1170.442,98.497,-52.091,-179.030,6.280,148.851
C01610=1170.438,98.746,-52.110,-179.028,6.281,148.850
C01611=1170.433,98.995,-52.128,-179.025,6.282,148.850
C01612=1170.428,99.245,-52.146,-179.022,6.284,148.849
C01613=1170.423,99.494,-52.165,-179.020,6.285,148.849
C01614=1170.418,99.743,-52.183,-179.016,6.286,148.848
C01615=1170.413,99.992,-52.201,-179.014,6.288,148.848
C01616=1170.409,100.242,-52.220,-179.012,6.289,148.847
C01617=1170.404,100.491,-52.238,-179.008,6.290,148.847
C01618=1170.398,100.740,-52.256,-179.006,6.291,148.846
C01619=1170.393,100.990,-52.274,-179.004,6.293,148.846
C01620=1170.389,101.239,-52.293,-179.000,6.294,148.845
C01621=1170.385,101.488,-52.311,-178.998,6.295,148.845
C01622=1170.379,101.737,-52.330,-178.995,6.297,148.844
C01623=1170.374,101.987,-52.348,-178.992,6.298,148.844
C01624=1170.370,102.236,-52.367,-178.990,6.299,148.843
C01625=1170.365,102.485,-52.385,-178.987,6.301,148.843
C01626=1170.359,102.735,-52.403,-178.984,6.302,148.842
C01627=1170.355,102.984,-52.422,-178.982,6.303,148.842
C01628=1170.351,103.233,-52.440,-178.979,6.305,148.841
C01629=1170.346,103.482,-52.458,-178.977,6.306,148.841
C01630=1170.340,103.732,-52.477,-178.974,6.307,148.840
C01631=1170.336,103.981,-52.496,-178.971,6.309,148.840
C01632=1170.331,104.230,-52.514,-178.969,6.310,148.840
C01633=1170.325,104.480,-52.533,-178.966,6.311,148.839
C01634=1170.321,104.729,-52.552,-178.963,6.312,148.839
C01635=1170.316,104.978,-52.570,-178.961,6.314,148.838
C01636=1170.311,105.227,-52.589,-178.958,6.315,148.837
C01637=1170.307,105.477,-52.607,-178.955,6.316,148.837
C01638=1170.302,105.726,-52.625,-178.953,6.318,148.837
C01639=1170.296,105.994,-52.646,-178.949,6.320,148.836
C01640=1170.291,106.262,-52.665,-178.947,6.321,148.836
C01641=1170.286,106.531,-52.686,-178.944,6.322,148.835
C01642=1170.281,106.799,-52.706,-178.941,6.324,148.835
C01643=1170.276,107.049,-52.724,-178.939,6.325,148.834
C01644=1170.272,107.298,-52.744,-178.935,6.327,148.834
C01645=1170.266,107.547,-52.762,-178.933,6.328,148.833
C01646=1170.261,107.796,-52.781,-178.930,6.329,148.833
C01647=1170.256,108.046,-52.800,-178.927,6.331,148.832
C01648=1170.252,108.295,-52.818,-178.925,6.332,148.832
C01649=1170.247,108.544,-52.837,-178.922,6.333,148.831
C01650=1170.242,108.793,-52.856,-178.920,6.335,148.831
C01651=1170.237,109.042,-52.874,-178.917,6.336,148.830
C01652=1170.232,109.292,-52.894,-178.914,6.337,148.830
C01653=1170.228,109.541,-52.912,-178.912,6.339,148.829
C01654=1170.223,109.791,-52.931,-178.908,6.340,148.829
C01655=1170.218,110.039,-52.950,-178.906,6.341,148.828
C01656=1170.213,110.289,-52.969,-178.904,6.343,148.828
C01657=1170.209,110.538,-52.988,-178.901,6.345,148.828
C01658=1170.203,110.787,-53.007,-178.898,6.346,148.827
C01659=1170.199,111.037,-53.025,-178.896,6.347,148.826
C01660=1170.194,111.286,-53.045,-178.893,6.349,148.826
C01661=1170.190,111.535,-53.064,-178.890,6.350,148.826
C01662=1170.184,111.784,-53.082,-178.888,6.351,148.825
C01663=1170.179,112.033,-53.101,-178.885,6.353,148.825
C01664=1170.175,112.283,-53.121,-178.882,6.354,148.824
C01665=1170.170,112.532,-53.139,-178.879,6.356,148.824
C01666=1170.165,112.781,-53.158,-178.877,6.357,148.823
C01667=1170.160,113.030,-53.177,-178.874,6.358,148.823
C01668=1170.155,113.280,-53.196,-178.871,6.360,148.822
C01669=1170.150,113.529,-53.215,-178.868,6.361,148.822
C01670=1170.146,113.778,-53.234,-178.866,6.362,148.821
C01671=1170.141,114.027,-53.254,-178.863,6.364,148.821
C01672=1170.137,114.276,-53.273,-178.861,6.366,148.821
C01673=1170.131,114.526,-53.291,-178.857,6.367,148.820
C01674=1170.126,114.775,-53.311,-178.855,6.368,148.819
C01675=1170.122,115.024,-53.329,-178.853,6.370,148.819
C01676=1170.117,115.274,-53.349,-178.850,6.371,148.819
C01677=1170.112,115.522,-53.368,-178.847,6.373,148.818
C01678=1170.107,115.772,-53.387,-178.845,6.374,148.818
C01679=1170.102,116.021,-53.406,-178.842,6.375,148.817
C01680=1170.098,116.270,-53.425,-178.839,6.377,148.817
C01681=1170.092,116.519,-53.444,-178.836,6.379,148.816
C01682=1170.088,116.769,-53.464,-178.834,6.379,148.816
C01683=1170.083,117.017,-53.483,-178.831,6.381,148.815
C01684=1170.078,117.267,-53.502,-178.828,6.383,148.815
C01685=1170.073,117.516,-53.521,-178.825,6.384,148.814
C01686=1170.068,117.766,-53.541,-178.823,6.385,148.814
C01687=1170.063,118.015,-53.559,-178.820,6.387,148.814
C01688=1170.059,118.264,-53.579,-178.818,6.389,148.813
C01689=1170.054,118.514,-53.599,-178.815,6.390,148.813
C01690=1170.049,118.762,-53.617,-178.812,6.391,148.812
C01691=1170.045,119.012,-53.637,-178.810,6.393,148.812
C01692=1170.039,119.261,-53.656,-178.807,6.394,148.811
C01693=1170.034,119.510,-53.676,-178.804,6.396,148.811
C01694=1170.030,119.759,-53.695,-178.801,6.397,148.810
C01695=1170.025,120.008,-53.714,-178.799,6.398,148.810
C01696=1170.020,120.258,-53.734,-178.796,6.400,148.809
C01697=1170.015,120.507,-53.753,-178.793,6.402,148.809
C01698=1170.011,120.756,-53.772,-178.791,6.404,148.809
C01699=1170.006,121.006,-53.792,-178.788,6.404,148.808
C01700=1170.001,121.254,-53.811,-178.785,6.406,148.808
C01701=1169.996,121.504,-53.831,-178.783,6.408,148.807
C01702=1169.991,121.753,-53.850,-178.780,6.409,148.807
C01703=1169.987,122.002,-53.870,-178.777,6.411,148.806
C01704=1169.982,122.251,-53.890,-178.775,6.412,148.806
C01705=1169.977,122.500,-53.909,-178.772,6.413,148.805
C01706=1169.972,122.750,-53.929,-178.769,6.415,148.805
C01707=1169.968,122.999,-53.948,-178.767,6.417,148.805
C01708=1169.962,123.248,-53.968,-178.763,6.418,148.804
C01709=1169.958,123.497,-53.987,-178.761,6.419,148.804
C01710=1169.954,123.746,-54.007,-178.759,6.421,148.803
C01711=1169.948,123.995,-54.026,-178.756,6.423,148.803
C01712=1169.944,124.245,-54.046,-178.753,6.424,148.802
C01713=1169.939,124.494,-54.066,-178.750,6.426,148.802
C01714=1169.934,124.743,-54.085,-178.748,6.427,148.801
C01715=1169.929,124.992,-54.105,-178.745,6.428,148.801
C01716=1169.924,125.242,-54.125,-178.742,6.430,148.801
C01717=1169.919,125.490,-54.144,-178.740,6.432,148.800
C01718=1169.915,125.740,-54.163,-178.737,6.433,148.800
C01719=1169.911,125.989,-54.184,-178.734,6.435,148.799
C01720=1169.906,126.238,-54.203,-178.732,6.436,148.799
C01721=1169.901,126.487,-54.223,-178.729,6.437,148.798
C01722=1169.896,126.737,-54.242,-178.726,6.439,148.798
C01723=1169.891,126.986,-54.263,-178.724,6.441,148.798
C01724=1169.886,127.234,-54.282,-178.720,6.442,148.797
C01725=1169.881,127.484,-54.302,-178.718,6.444,148.797
C01726=1169.877,127.733,-54.322,-178.716,6.445,148.796
C01727=1169.872,127.983,-54.342,-178.713,6.447,148.796
C01728=1169.867,128.231,-54.361,-178.710,6.448,148.795
C01729=1169.862,128.480,-54.381,-178.707,6.450,148.795
C01730=1169.858,128.730,-54.401,-178.704,6.452,148.794
C01731=1169.853,128.979,-54.421,-178.702,6.453,148.794
C01732=1169.848,129.228,-54.441,-178.699,6.454,148.794
C01733=1169.843,129.477,-54.460,-178.697,6.456,148.793
C01734=1169.839,129.726,-54.481,-178.694,6.458,148.793
C01735=1169.834,129.976,-54.500,-178.691,6.459,148.792
C01736=1169.829,130.225,-54.521,-178.688,6.461,148.792
C01737=1169.824,130.474,-54.540,-178.685,6.463,148.791
C01738=1169.820,130.723,-54.560,-178.683,6.464,148.791
C01739=1169.814,130.973,-54.581,-178.681,6.465,148.791
C01740=1169.810,131.221,-54.601,-178.678,6.467,148.790
C01741=1169.805,131.471,-54.621,-178.675,6.469,148.790
C01742=1169.800,131.719,-54.641,-178.672,6.470,148.789
C01743=1169.795,131.988,-54.662,-178.669,6.472,148.789
C01744=1169.789,132.257,-54.683,-178.667,6.473,148.788
C01745=1169.785,132.525,-54.705,-178.663,6.475,148.788
C01746=1169.779,132.794,-54.727,-178.661,6.477,148.787
C01747=1169.775,133.043,-54.747,-178.658,6.478,148.787
C01748=1169.770,133.292,-54.767,-178.655,6.480,148.787
C01749=1169.765,133.541,-54.787,-178.653,6.482,148.786
C01750=1169.761,133.791,-54.807,-178.650,6.484,148.786
C01751=1169.756,134.040,-54.827,-178.647,6.485,148.785
C01752=1169.750,134.289,-54.847,-178.644,6.487,148.785
C01753=1169.746,134.538,-54.868,-178.642,6.488,148.784
C01754=1169.741,134.787,-54.888,-178.639,6.489,148.784
C01755=1169.737,135.036,-54.908,-178.636,6.491,148.784
C01756=1169.732,135.285,-54.928,-178.634,6.493,148.783
C01757=1169.727,135.535,-54.949,-178.631,6.495,148.783
C01758=1169.722,135.784,-54.969,-178.628,6.496,148.782
C01759=1169.718,136.033,-54.989,-178.625,6.498,148.782
C01760=1169.713,136.281,-55.009,-178.622,6.499,148.781
C01761=1169.708,136.531,-55.030,-178.620,6.501,148.781
C01762=1169.703,136.780,-55.050,-178.618,6.502,148.781
C01763=1169.698,137.029,-55.070,-178.615,6.504,148.780
C01764=1169.694,137.278,-55.090,-178.612,6.506,148.780
C01765=1169.689,137.527,-55.111,-178.610,6.507,148.780
C01766=1169.684,137.777,-55.131,-178.607,6.509,148.779
C01767=1169.680,138.026,-55.151,-178.604,6.510,148.779
C01768=1169.675,138.275,-55.172,-178.601,6.512,148.778
C01769=1169.670,138.524,-55.193,-178.598,6.514,148.778
C01770=1169.665,138.774,-55.212,-178.596,6.516,148.777
C01771=1169.661,139.023,-55.233,-178.593,6.517,148.777
C01772=1169.656,139.272,-55.254,-178.590,6.519,148.777
C01773=1169.651,139.521,-55.274,-178.588,6.520,148.776
C01774=1169.647,139.770,-55.294,-178.585,6.522,148.776
C01775=1169.642,140.019,-55.315,-178.583,6.523,148.775
C01776=1169.637,140.267,-55.335,-178.580,6.525,148.775
C01777=1169.632,140.517,-55.355,-178.577,6.527,148.774
C01778=1169.627,140.766,-55.376,-178.574,6.528,148.774
C01779=1169.622,141.015,-55.396,-178.571,6.530,148.774
C01780=1169.617,141.264,-55.417,-178.569,6.532,148.773
C01781=1169.613,141.513,-55.438,-178.566,6.534,148.773
C01782=1169.608,141.762,-55.458,-178.563,6.535,148.772
C01783=1169.603,142.012,-55.479,-178.561,6.537,148.772
C01784=1169.599,142.260,-55.499,-178.558,6.539,148.772
C01785=1169.594,142.509,-55.520,-178.555,6.541,148.771
C01786=1169.590,142.759,-55.541,-178.552,6.542,148.771
C01787=1169.585,143.008,-55.561,-178.550,6.543,148.771
C01788=1169.580,143.258,-55.582,-178.548,6.545,148.770
C01789=1169.575,143.507,-55.603,-178.544,6.546,148.770
C01790=1169.570,143.756,-55.624,-178.542,6.548,148.769
C01791=1169.566,144.005,-55.644,-178.539,6.550,148.769
C01792=1169.561,144.254,-55.665,-178.536,6.552,148.768
C01793=1169.556,144.503,-55.685,-178.534,6.553,148.768
C01794=1169.551,144.752,-55.706,-178.531,6.555,148.768
C01795=1169.547,145.001,-55.727,-178.528,6.557,148.767
C01796=1169.543,145.250,-55.748,-178.526,6.559,148.767
C01797=1169.537,145.499,-55.769,-178.523,6.560,148.766
C01798=1169.532,145.748,-55.790,-178.520,6.562,148.766
C01799=1169.528,145.997,-55.810,-178.517,6.564,148.766
C01800=1169.523,146.246,-55.831,-178.515,6.566,148.765
C01801=1169.518,146.495,-55.852,-178.512,6.567,148.765
C01802=1169.514,146.745,-55.873,-178.509,6.569,148.765
C01803=1169.509,146.994,-55.893,-178.507,6.571,148.764
C01804=1169.504,147.243,-55.915,-178.504,6.572,148.764
C01805=1169.500,147.492,-55.935,-178.501,6.574,148.763
C01806=1169.495,147.741,-55.956,-178.498,6.576,148.763
C01807=1169.490,147.990,-55.977,-178.495,6.577,148.762
C01808=1169.485,148.239,-55.998,-178.493,6.579,148.762
C01809=1169.480,148.488,-56.019,-178.490,6.581,148.762
C01810=1169.476,148.737,-56.040,-178.487,6.583,148.761
C01811=1169.471,148.987,-56.061,-178.485,6.584,148.761
C01812=1169.467,149.235,-56.082,-178.482,6.586,148.761
C01813=1169.462,149.484,-56.103,-178.479,6.588,148.760
C01814=1169.457,149.734,-56.124,-178.477,6.590,148.760
C01815=1169.452,149.983,-56.144,-178.474,6.591,148.759
C01816=1169.447,150.231,-56.166,-178.471,6.593,148.759
C01817=1169.443,150.481,-56.187,-178.468,6.595,148.759
C01818=1169.438,150.730,-56.208,-178.466,6.597,148.758
C01819=1169.433,150.979,-56.229,-178.463,6.598,148.758
C01820=1169.428,151.228,-56.250,-178.460,6.600,148.757
C01821=1169.424,151.477,-56.271,-178.458,6.602,148.757
C01822=1169.419,151.726,-56.292,-178.455,6.604,148.757
C01823=1169.414,151.976,-56.314,-178.452,6.605,148.756
C01824=1169.410,152.224,-56.335,-178.450,6.607,148.756
C01825=1169.405,152.473,-56.356,-178.447,6.609,148.756
C01826=1169.400,152.722,-56.377,-178.444,6.611,148.755
C01827=1169.395,152.971,-56.398,-178.441,6.612,148.755
C01828=1169.391,153.221,-56.419,-178.439,6.614,148.754
C01829=1169.386,153.469,-56.441,-178.436,6.616,148.754
C01830=1169.381,153.719,-56.462,-178.433,6.618,148.754
C01831=1169.376,153.967,-56.484,-178.431,6.619,148.753
C01832=1169.372,154.217,-56.505,-178.428,6.621,148.753
C01833=1169.368,154.465,-56.526,-178.425,6.623,148.753
C01834=1169.362,154.715,-56.547,-178.423,6.625,148.752
C01835=1169.358,154.963,-56.569,-178.420,6.626,148.752
C01836=1169.353,155.213,-56.590,-178.417,6.628,148.751
C01837=1169.349,155.462,-56.611,-178.415,6.630,148.751
C01838=1169.344,155.711,-56.632,-178.412,6.632,148.751
